LIN {X 0,Y 450.155,Z 511.876,A -85,B 0,C 180,E1 -8846.56,E2 -8846.56} C_VEL
LIN {X 0,Y 446.595,Z 503.795,A -85,B 0,C 180,E1 -8847.024,E2 -8847.024} C_VEL
LIN {X 0,Y 446.473,Z 503.185,A -85,B 0,C 180,E1 -8847.064,E2 -8847.064} C_VEL
LIN {X 0,Y 446.432,Z 503.191,A -85,B 0,C 180,E1 -8850.25,E2 -8850.25} C_VEL
LIN {X 0,Y 446.45,Z 503.188,A -85,B 0,C 180,E1 -8853.454,E2 -8853.454} C_VEL
LIN {X 0,Y 446.414,Z 503.19,A -85,B 0,C 180,E1 -8856.745,E2 -8856.745} C_VEL
LIN {X 0,Y 446.46,Z 503.185,A -85,B 0,C 180,E1 -8859.525,E2 -8859.525} C_VEL
LIN {X 0,Y 446.434,Z 503.188,A -85,B 0,C 180,E1 -8862.605,E2 -8862.605} C_VEL
LIN {X 0,Y 446.457,Z 503.185,A -85,B 0,C 180,E1 -8865.104,E2 -8865.104} C_VEL
LIN {X 0,Y 446.434,Z 503.189,A -85,B 0,C 180,E1 -8868.609,E2 -8868.609} C_VEL
LIN {X 0,Y 446.465,Z 503.184,A -85,B 0,C 180,E1 -8870.975,E2 -8870.975} C_VEL
LIN {X 0,Y 446.425,Z 503.194,A -85,B 0,C 180,E1 -8874.374,E2 -8874.374} C_VEL
LIN {X 0,Y 446.428,Z 503.194,A -85,B 0,C 180,E1 -8877.638,E2 -8877.638} C_VEL
LIN {X 0,Y 446.454,Z 503.189,A -85,B 0,C 180,E1 -8880.79,E2 -8880.79} C_VEL
LIN {X 0,Y 446.603,Z 503.368,A -85,B 0,C 180,E1 -8884.357,E2 -8884.357} C_VEL
LIN {X 0,Y 446.829,Z 506.002,A -85,B 0,C 180,E1 -8885.861,E2 -8885.861} C_VEL
LIN {X 0,Y 446.728,Z 511.144,A -85,B 0,C 180,E1 -8888.786,E2 -8888.786} C_VEL
LIN {X 0,Y 446.692,Z 516.086,A -85,B 0,C 180,E1 -8891.658,E2 -8891.658} C_VEL
LIN {X 0,Y 446.583,Z 520.857,A -85,B 0,C 180,E1 -8894.482,E2 -8894.482} C_VEL
LIN {X 0,Y 446.532,Z 523.772,A -85,B 0,C 180,E1 -8896.223,E2 -8896.223} C_VEL
LIN {X 0,Y 446.518,Z 525.315,A -85,B 0,C 180,E1 -8896.662,E2 -8896.662} C_VEL
LIN {X 0,Y 446.485,Z 527.885,A -85,B 0,C 180,E1 -8897.023,E2 -8897.023} C_VEL
LIN {X 0,Y 446.494,Z 532.862,A -85,B 0,C 180,E1 -8897.431,E2 -8897.431} C_VEL
LIN {X 0,Y 446.761,Z 538.729,A -85,B 0,C 180,E1 -8897.718,E2 -8897.718} C_VEL
LIN {X 0,Y 448.261,Z 548.9,A -85,B 0,C 180,E1 -8898.125,E2 -8898.125} C_VEL
LIN {X 0,Y 448.835,Z 550.834,A -85,B 0,C 180,E1 -8898.219,E2 -8898.219} C_VEL
LIN {X 0,Y 451.313,Z 559.337,A -85,B 0,C 180,E1 -8898.674,E2 -8898.674} C_VEL
LIN {X 0,Y 450.413,Z 575.184,A -85,B 0,C 180,E1 -8899.321,E2 -8899.321} C_VEL
LIN {X 0,Y 449.401,Z 589.936,A -85,B 0,C 180,E1 -8900.094,E2 -8900.094} C_VEL
LIN {X 0,Y 448.277,Z 603.783,A -85,B 0,C 180,E1 -8900.979,E2 -8900.979} C_VEL
LIN {X 0,Y 446.836,Z 619.369,A -85,B 0,C 180,E1 -8902.203,E2 -8902.203} C_VEL
LIN {X 0,Y 445.504,Z 632.325,A -85,B 0,C 180,E1 -8903.432,E2 -8903.432} C_VEL
LIN {X 0,Y 444.217,Z 644.41,A -85,B 0,C 180,E1 -8904.78,E2 -8904.78} C_VEL
LIN {X 0,Y 442.907,Z 656.466,A -85,B 0,C 180,E1 -8906.36,E2 -8906.36} C_VEL
LIN {X 0,Y 441.78,Z 666.782,A -85,B 0,C 180,E1 -8907.948,E2 -8907.948} C_VEL
LIN {X 0,Y 440.691,Z 676.755,A -85,B 0,C 180,E1 -8909.771,E2 -8909.771} C_VEL
LIN {X 0,Y 439.993,Z 684.187,A -85,B 0,C 180,E1 -8911.372,E2 -8911.372} C_VEL
LIN {X 0,Y 439.339,Z 691.448,A -85,B 0,C 180,E1 -8913.209,E2 -8913.209} C_VEL
LIN {X 0,Y 438.864,Z 698.729,A -85,B 0,C 180,E1 -8915.513,E2 -8915.513} C_VEL
LIN {X 0,Y 438.632,Z 703.269,A -85,B 0,C 180,E1 -8917.363,E2 -8917.363} C_VEL
LIN {X 0,Y 438.377,Z 706.848,A -85,B 0,C 180,E1 -8919.224,E2 -8919.224} C_VEL
LIN {X 0,Y 438.327,Z 709.385,A -85,B 0,C 180,E1 -8921.092,E2 -8921.092} C_VEL
LIN {X 0,Y 438.225,Z 710.957,A -85,B 0,C 180,E1 -8922.974,E2 -8922.974} C_VEL
LIN {X 0,Y 438.204,Z 711.571,A -85,B 0,C 180,E1 -8924.868,E2 -8924.868} C_VEL
LIN {X 0,Y 438.165,Z 711.15,A -85,B 0,C 180,E1 -8926.78,E2 -8926.78} C_VEL
LIN {X 0,Y 438.249,Z 709.566,A -85,B 0,C 180,E1 -8928.886,E2 -8928.886} C_VEL
LIN {X 0,Y 438.342,Z 707.239,A -85,B 0,C 180,E1 -8930.653,E2 -8930.653} C_VEL
LIN {X 0,Y 438.597,Z 703.612,A -85,B 0,C 180,E1 -8932.616,E2 -8932.616} C_VEL
LIN {X 0,Y 438.891,Z 698.778,A -85,B 0,C 180,E1 -8934.602,E2 -8934.602} C_VEL
LIN {X 0,Y 439.358,Z 692.513,A -85,B 0,C 180,E1 -8936.607,E2 -8936.607} C_VEL
LIN {X 0,Y 439.992,Z 684.737,A -85,B 0,C 180,E1 -8938.631,E2 -8938.631} C_VEL
LIN {X 0,Y 440.894,Z 675.565,A -85,B 0,C 180,E1 -8940.595,E2 -8940.595} C_VEL
LIN {X 0,Y 441.839,Z 666.752,A -85,B 0,C 180,E1 -8942.194,E2 -8942.194} C_VEL
LIN {X 0,Y 443.121,Z 655.256,A -85,B 0,C 180,E1 -8943.957,E2 -8943.957} C_VEL
LIN {X 0,Y 444.545,Z 642.016,A -85,B 0,C 180,E1 -8945.658,E2 -8945.658} C_VEL
LIN {X 0,Y 446.007,Z 628.866,A -85,B 0,C 180,E1 -8947.064,E2 -8947.064} C_VEL
LIN {X 0,Y 447.418,Z 614.816,A -85,B 0,C 180,E1 -8948.325,E2 -8948.325} C_VEL
LIN {X 0,Y 448.686,Z 600.827,A -85,B 0,C 180,E1 -8949.372,E2 -8949.372} C_VEL
LIN {X 0,Y 449.83,Z 586.318,A -85,B 0,C 180,E1 -8950.27,E2 -8950.27} C_VEL
LIN {X 0,Y 450.93,Z 570.329,A -85,B 0,C 180,E1 -8951.057,E2 -8951.057} C_VEL
LIN {X 0,Y 451.396,Z 558.681,A -85,B 0,C 180,E1 -8951.513,E2 -8951.513} C_VEL
LIN {X 0,Y 447.422,Z 546.372,A -85,B 0,C 180,E1 -8952.201,E2 -8952.201} C_VEL
LIN {X 0,Y 440.677,Z 529.846,A -85,B 0,C 180,E1 -8953.077,E2 -8953.077} C_VEL
LIN {X 0,Y 439.565,Z 526.832,A -85,B 0,C 180,E1 -8953.229,E2 -8953.229} C_VEL
LIN {X 0,Y 439.698,Z 521.329,A -85,B 0,C 180,E1 -8956.583,E2 -8956.583} C_VEL
LIN {X 0,Y 439.823,Z 517.224,A -85,B 0,C 180,E1 -8959.069,E2 -8959.069} C_VEL
LIN {X 0,Y 439.901,Z 513.154,A -85,B 0,C 180,E1 -8961.519,E2 -8961.519} C_VEL
LIN {X 0,Y 439.979,Z 509.374,A -85,B 0,C 180,E1 -8963.77,E2 -8963.77} C_VEL
LIN {X 0,Y 439.715,Z 505.572,A -85,B 0,C 180,E1 -8965.985,E2 -8965.985} C_VEL
LIN {X 0,Y 439.39,Z 504.071,A -85,B 0,C 180,E1 -8966.949,E2 -8966.949} C_VEL
LIN {X 0,Y 439.389,Z 504.069,A -85,B 0,C 180,E1 -8970.274,E2 -8970.274} C_VEL
LIN {X 0,Y 439.425,Z 504.062,A -85,B 0,C 180,E1 -8973.587,E2 -8973.587} C_VEL
LIN {X 0,Y 439.38,Z 504.067,A -85,B 0,C 180,E1 -8976.429,E2 -8976.429} C_VEL
LIN {X 0,Y 439.384,Z 504.068,A -85,B 0,C 180,E1 -8979.396,E2 -8979.396} C_VEL
LIN {X 0,Y 439.422,Z 504.063,A -85,B 0,C 180,E1 -8982.309,E2 -8982.309} C_VEL
LIN {X 0,Y 439.438,Z 504.06,A -85,B 0,C 180,E1 -8985.173,E2 -8985.173} C_VEL
LIN {X 0,Y 439.498,Z 504.053,A -85,B 0,C 180,E1 -8988.001,E2 -8988.001} C_VEL
LIN {X 0,Y 439.537,Z 504.043,A -85,B 0,C 180,E1 -8991.726,E2 -8991.726} C_VEL
LIN {X 0,Y 439.619,Z 504.035,A -85,B 0,C 180,E1 -8994.495,E2 -8994.495} C_VEL
LIN {X 0,Y 439.626,Z 504.031,A -85,B 0,C 180,E1 -8998.167,E2 -8998.167} C_VEL
LIN {X 0,Y 439.754,Z 504.021,A -85,B 0,C 180,E1 -9000,E2 -9000} C_VEL
LIN {X 0,Y 439.647,Z 504.031,A -85,B 0,C 180,E1 -9002.748,E2 -9002.748} C_VEL
LIN {X 0,Y 439.607,Z 504.038,A -85,B 0,C 180,E1 -9006.425,E2 -9006.425} C_VEL
LIN {X 0,Y 439.491,Z 504.047,A -85,B 0,C 180,E1 -9009.201,E2 -9009.201} C_VEL
LIN {X 0,Y 439.493,Z 504.046,A -85,B 0,C 180,E1 -9012.727,E2 -9012.727} C_VEL
LIN {X 0,Y 439.435,Z 504.045,A -85,B 0,C 180,E1 -9016.349,E2 -9016.349} C_VEL
LIN {X 0,Y 439.423,Z 504.053,A -85,B 0,C 180,E1 -9019.625,E2 -9019.625} C_VEL
LIN {X 0,Y 439.366,Z 504.062,A -85,B 0,C 180,E1 -9022.575,E2 -9022.575} C_VEL
LIN {X 0,Y 439.401,Z 504.046,A -85,B 0,C 180,E1 -9025.585,E2 -9025.585} C_VEL
LIN {X 0,Y 439.414,Z 504.063,A -85,B 0,C 180,E1 -9028.673,E2 -9028.673} C_VEL
LIN {X 0,Y 439.372,Z 504.069,A -85,B 0,C 180,E1 -9032.034,E2 -9032.034} C_VEL
LIN {X 0,Y 439.386,Z 504.064,A -85,B 0,C 180,E1 -9035.341,E2 -9035.341} C_VEL
LIN {X 0,Y 439.391,Z 504.064,A -85,B 0,C 180,E1 -9038.594,E2 -9038.594} C_VEL
LIN {X 0,Y 439.425,Z 504.199,A -85,B 0,C 180,E1 -9040.749,E2 -9040.749} C_VEL
LIN {X 0,Y 441.305,Z 512.586,A -85,B 0,C 180,E1 -9043.757,E2 -9043.757} C_VEL
LIN {X 0,Y 443.373,Z 522.19,A -85,B 0,C 180,E1 -9047.033,E2 -9047.033} C_VEL
LIN {X 0,Y 444.482,Z 528.015,A -85,B 0,C 180,E1 -9048.937,E2 -9048.937} C_VEL
LIN {X 0,Y 444.326,Z 534.065,A -85,B 0,C 180,E1 -9050.753,E2 -9050.753} C_VEL
LIN {X 0,Y 443.528,Z 545.656,A -85,B 0,C 180,E1 -9054.108,E2 -9054.108} C_VEL
LIN {X 0,Y 442.749,Z 557.216,A -85,B 0,C 180,E1 -9057.338,E2 -9057.338} C_VEL
LIN {X 0,Y 441.923,Z 570.71,A -85,B 0,C 180,E1 -9061.006,E2 -9061.006} C_VEL
LIN {X 0,Y 441.695,Z 574.164,A -85,B 0,C 180,E1 -9061.932,E2 -9061.932} C_VEL
LIN {X 0,Y 447.617,Z 596.261,A -85,B 0,C 180,E1 -9062.818,E2 -9062.818} C_VEL
LIN {X 0,Y 451.098,Z 610.608,A -85,B 0,C 180,E1 -9063.501,E2 -9063.501} C_VEL
LIN {X 0,Y 450.151,Z 626.715,A -85,B 0,C 180,E1 -9064.141,E2 -9064.141} C_VEL
LIN {X 0,Y 448.858,Z 643.305,A -85,B 0,C 180,E1 -9064.993,E2 -9064.993} C_VEL
LIN {X 0,Y 447.49,Z 659.254,A -85,B 0,C 180,E1 -9066.024,E2 -9066.024} C_VEL
LIN {X 0,Y 446.086,Z 673.924,A -85,B 0,C 180,E1 -9067.174,E2 -9067.174} C_VEL
LIN {X 0,Y 444.736,Z 687.558,A -85,B 0,C 180,E1 -9068.445,E2 -9068.445} C_VEL
LIN {X 0,Y 443.475,Z 700.18,A -85,B 0,C 180,E1 -9069.839,E2 -9069.839} C_VEL
LIN {X 0,Y 442.164,Z 712.75,A -85,B 0,C 180,E1 -9071.466,E2 -9071.466} C_VEL
LIN {X 0,Y 441.22,Z 722.902,A -85,B 0,C 180,E1 -9072.999,E2 -9072.999} C_VEL
LIN {X 0,Y 440.324,Z 732.743,A -85,B 0,C 180,E1 -9074.732,E2 -9074.732} C_VEL
LIN {X 0,Y 439.596,Z 741.658,A -85,B 0,C 180,E1 -9076.597,E2 -9076.597} C_VEL
LIN {X 0,Y 439.076,Z 749.128,A -85,B 0,C 180,E1 -9078.46,E2 -9078.46} C_VEL
LIN {X 0,Y 438.661,Z 755.325,A -85,B 0,C 180,E1 -9080.316,E2 -9080.316} C_VEL
LIN {X 0,Y 438.495,Z 760.18,A -85,B 0,C 180,E1 -9082.171,E2 -9082.171} C_VEL
LIN {X 0,Y 438.394,Z 763.307,A -85,B 0,C 180,E1 -9083.685,E2 -9083.685} C_VEL
LIN {X 0,Y 438.286,Z 765.978,A -85,B 0,C 180,E1 -9085.402,E2 -9085.402} C_VEL
LIN {X 0,Y 438.282,Z 767.896,A -85,B 0,C 180,E1 -9087.244,E2 -9087.244} C_VEL
LIN {X 0,Y 438.226,Z 768.847,A -85,B 0,C 180,E1 -9089.082,E2 -9089.082} C_VEL
LIN {X 0,Y 438.226,Z 768.847,A -85,B 0,C 180,E1 -9090.92,E2 -9090.92} C_VEL
LIN {X 0,Y 438.282,Z 767.893,A -85,B 0,C 180,E1 -9092.758,E2 -9092.758} C_VEL
LIN {X 0,Y 438.287,Z 765.974,A -85,B 0,C 180,E1 -9094.6,E2 -9094.6} C_VEL
LIN {X 0,Y 438.418,Z 763.059,A -85,B 0,C 180,E1 -9096.444,E2 -9096.444} C_VEL
LIN {X 0,Y 438.535,Z 759.098,A -85,B 0,C 180,E1 -9098.294,E2 -9098.294} C_VEL
LIN {X 0,Y 438.71,Z 753.832,A -85,B 0,C 180,E1 -9100.15,E2 -9100.15} C_VEL
LIN {X 0,Y 439.198,Z 747.328,A -85,B 0,C 180,E1 -9102.007,E2 -9102.007} C_VEL
LIN {X 0,Y 439.752,Z 739.357,A -85,B 0,C 180,E1 -9103.871,E2 -9103.871} C_VEL
LIN {X 0,Y 440.586,Z 729.818,A -85,B 0,C 180,E1 -9105.735,E2 -9105.735} C_VEL
LIN {X 0,Y 441.45,Z 719.525,A -85,B 0,C 180,E1 -9107.438,E2 -9107.438} C_VEL
LIN {X 0,Y 442.487,Z 708.476,A -85,B 0,C 180,E1 -9109.003,E2 -9109.003} C_VEL
LIN {X 0,Y 443.699,Z 695.677,A -85,B 0,C 180,E1 -9110.546,E2 -9110.546} C_VEL
LIN {X 0,Y 445.098,Z 681.138,A -85,B 0,C 180,E1 -9112.025,E2 -9112.025} C_VEL
LIN {X 0,Y 446.476,Z 666.202,A -85,B 0,C 180,E1 -9113.298,E2 -9113.298} C_VEL
LIN {X 0,Y 447.827,Z 650.15,A -85,B 0,C 180,E1 -9114.434,E2 -9114.434} C_VEL
LIN {X 0,Y 449.261,Z 632.83,A -85,B 0,C 180,E1 -9115.419,E2 -9115.419} C_VEL
LIN {X 0,Y 450.375,Z 616.592,A -85,B 0,C 180,E1 -9116.155,E2 -9116.155} C_VEL
LIN {X 0,Y 450.617,Z 609.71,A -85,B 0,C 180,E1 -9116.429,E2 -9116.429} C_VEL
LIN {X 0,Y 446.065,Z 591.603,A -85,B 0,C 180,E1 -9117.299,E2 -9117.299} C_VEL
LIN {X 0,Y 441.305,Z 569.539,A -85,B 0,C 180,E1 -9118.175,E2 -9118.175} C_VEL
LIN {X 0,Y 441.748,Z 557.378,A -85,B 0,C 180,E1 -9121.169,E2 -9121.169} C_VEL
LIN {X 0,Y 442.142,Z 544.142,A -85,B 0,C 180,E1 -9124.532,E2 -9124.532} C_VEL
LIN {X 0,Y 442.565,Z 534.404,A -85,B 0,C 180,E1 -9127.118,E2 -9127.118} C_VEL
LIN {X 0,Y 443.037,Z 524.605,A -85,B 0,C 180,E1 -9129.895,E2 -9129.895} C_VEL
LIN {X 0,Y 442.696,Z 520.674,A -85,B 0,C 180,E1 -9131.139,E2 -9131.139} C_VEL
LIN {X 0,Y 441.448,Z 513.639,A -85,B 0,C 180,E1 -9133.692,E2 -9133.692} C_VEL
LIN {X 0,Y 440.452,Z 508.687,A -85,B 0,C 180,E1 -9135.893,E2 -9135.893} C_VEL
LIN {X 0,Y 439.43,Z 504.239,A -85,B 0,C 180,E1 -9138.57,E2 -9138.57} C_VEL
LIN {X 0,Y 439.386,Z 504.068,A -85,B 0,C 180,E1 -9141.607,E2 -9141.607} C_VEL
LIN {X 0,Y 439.402,Z 504.065,A -85,B 0,C 180,E1 -9144.845,E2 -9144.845} C_VEL
LIN {X 0,Y 439.374,Z 504.069,A -85,B 0,C 180,E1 -9148.14,E2 -9148.14} C_VEL
LIN {X 0,Y 439.434,Z 504.061,A -85,B 0,C 180,E1 -9151.599,E2 -9151.599} C_VEL
LIN {X 0,Y 439.421,Z 504.063,A -85,B 0,C 180,E1 -9152.387,E2 -9152.387} C_VEL
LIN {X 0,Y 440.516,Z 507.043,A -85,B 0,C 180,E1 -9152.569,E2 -9152.569} C_VEL
LIN {X 0,Y 446.024,Z 518.302,A -85,B 0,C 180,E1 -9153.371,E2 -9153.371} C_VEL
LIN {X 0,Y 449.995,Z 528.652,A -85,B 0,C 180,E1 -9154.069,E2 -9154.069} C_VEL
LIN {X 0,Y 450.431,Z 530.462,A -85,B 0,C 180,E1 -9154.184,E2 -9154.184} C_VEL
LIN {X 0,Y 449.563,Z 546.73,A -85,B 0,C 180,E1 -9154.952,E2 -9154.952} C_VEL
LIN {X 0,Y 448.392,Z 562.457,A -85,B 0,C 180,E1 -9155.877,E2 -9155.877} C_VEL
LIN {X 0,Y 447.292,Z 576.15,A -85,B 0,C 180,E1 -9156.871,E2 -9156.871} C_VEL
LIN {X 0,Y 446.14,Z 589.85,A -85,B 0,C 180,E1 -9158.054,E2 -9158.054} C_VEL
LIN {X 0,Y 444.907,Z 602.248,A -85,B 0,C 180,E1 -9159.313,E2 -9159.313} C_VEL
LIN {X 0,Y 443.843,Z 612.936,A -85,B 0,C 180,E1 -9160.578,E2 -9160.578} C_VEL
LIN {X 0,Y 442.707,Z 624.177,A -85,B 0,C 180,E1 -9162.141,E2 -9162.141} C_VEL
LIN {X 0,Y 441.682,Z 634.47,A -85,B 0,C 180,E1 -9163.832,E2 -9163.832} C_VEL
LIN {X 0,Y 440.75,Z 643.955,A -85,B 0,C 180,E1 -9165.691,E2 -9165.691} C_VEL
LIN {X 0,Y 440.064,Z 651.852,A -85,B 0,C 180,E1 -9167.55,E2 -9167.55} C_VEL
LIN {X 0,Y 439.461,Z 658.362,A -85,B 0,C 180,E1 -9169.403,E2 -9169.403} C_VEL
LIN {X 0,Y 439.057,Z 664.718,A -85,B 0,C 180,E1 -9171.717,E2 -9171.717} C_VEL
LIN {X 0,Y 438.809,Z 668.498,A -85,B 0,C 180,E1 -9173.563,E2 -9173.563} C_VEL
LIN {X 0,Y 438.609,Z 671.321,A -85,B 0,C 180,E1 -9175.405,E2 -9175.405} C_VEL
LIN {X 0,Y 438.529,Z 673.1,A -85,B 0,C 180,E1 -9177.245,E2 -9177.245} C_VEL
LIN {X 0,Y 438.445,Z 673.979,A -85,B 0,C 180,E1 -9179.082,E2 -9179.082} C_VEL
LIN {X 0,Y 438.432,Z 673.872,A -85,B 0,C 180,E1 -9180.919,E2 -9180.919} C_VEL
LIN {X 0,Y 438.527,Z 672.857,A -85,B 0,C 180,E1 -9182.756,E2 -9182.756} C_VEL
LIN {X 0,Y 438.58,Z 670.871,A -85,B 0,C 180,E1 -9184.596,E2 -9184.596} C_VEL
LIN {X 0,Y 438.77,Z 667.318,A -85,B 0,C 180,E1 -9186.74,E2 -9186.74} C_VEL
LIN {X 0,Y 438.973,Z 662.731,A -85,B 0,C 180,E1 -9188.749,E2 -9188.749} C_VEL
LIN {X 0,Y 439.245,Z 657.369,A -85,B 0,C 180,E1 -9190.603,E2 -9190.603} C_VEL
LIN {X 0,Y 439.811,Z 650.68,A -85,B 0,C 180,E1 -9192.458,E2 -9192.458} C_VEL
LIN {X 0,Y 440.454,Z 642.654,A -85,B 0,C 180,E1 -9194.32,E2 -9194.32} C_VEL
LIN {X 0,Y 441.227,Z 634.366,A -85,B 0,C 180,E1 -9195.948,E2 -9195.948} C_VEL
LIN {X 0,Y 442.149,Z 624.564,A -85,B 0,C 180,E1 -9197.579,E2 -9197.579} C_VEL
LIN {X 0,Y 443.238,Z 613.092,A -85,B 0,C 180,E1 -9199.209,E2 -9199.209} C_VEL
LIN {X 0,Y 444.544,Z 600.249,A -85,B 0,C 180,E1 -9200.75,E2 -9200.75} C_VEL
LIN {X 0,Y 445.85,Z 586.862,A -85,B 0,C 180,E1 -9202.108,E2 -9202.108} C_VEL
LIN {X 0,Y 447.029,Z 573.338,A -85,B 0,C 180,E1 -9203.267,E2 -9203.267} C_VEL
LIN {X 0,Y 448.267,Z 558.807,A -85,B 0,C 180,E1 -9204.3,E2 -9204.3} C_VEL
LIN {X 0,Y 449.287,Z 544.247,A -85,B 0,C 180,E1 -9205.16,E2 -9205.16} C_VEL
LIN {X 0,Y 450.169,Z 530.335,A -85,B 0,C 180,E1 -9205.83,E2 -9205.83} C_VEL
LIN {X 0,Y 445.202,Z 517.627,A -85,B 0,C 180,E1 -9206.658,E2 -9206.658} C_VEL
LIN {X 0,Y 439.48,Z 504.426,A -85,B 0,C 180,E1 -9207.46,E2 -9207.46} C_VEL
LIN {X 0,Y 439.429,Z 504.06,A -85,B 0,C 180,E1 -9207.493,E2 -9207.493} C_VEL
LIN {X 0,Y 439.366,Z 504.07,A -85,B 0,C 180,E1 -9210.789,E2 -9210.789} C_VEL
LIN {X 0,Y 439.393,Z 504.065,A -85,B 0,C 180,E1 -9214.044,E2 -9214.044} C_VEL
LIN {X 0,Y 439.362,Z 504.069,A -85,B 0,C 180,E1 -9216.889,E2 -9216.889} C_VEL
LIN {X 0,Y 439.407,Z 504.064,A -85,B 0,C 180,E1 -9219.849,E2 -9219.849} C_VEL
LIN {X 0,Y 439.387,Z 504.066,A -85,B 0,C 180,E1 -9222.627,E2 -9222.627} C_VEL
LIN {X 0,Y 439.405,Z 504.063,A -85,B 0,C 180,E1 -9225.271,E2 -9225.271} C_VEL
LIN {X 0,Y 439.394,Z 504.067,A -85,B 0,C 180,E1 -9228.743,E2 -9228.743} C_VEL
LIN {X 0,Y 439.383,Z 504.069,A -85,B 0,C 180,E1 -9231.607,E2 -9231.607} C_VEL
LIN {X 0,Y 439.405,Z 504.066,A -85,B 0,C 180,E1 -9234.844,E2 -9234.844} C_VEL
LIN {X 0,Y 439.379,Z 504.072,A -85,B 0,C 180,E1 -9238.139,E2 -9238.139} C_VEL
LIN {X 0,Y 439.438,Z 504.063,A -85,B 0,C 180,E1 -9241.598,E2 -9241.598} C_VEL
LIN {X 0,Y 439.488,Z 504.068,A -85,B 0,C 180,E1 -9244.05,E2 -9244.05} C_VEL
LIN {X 0,Y 439.794,Z 508.249,A -85,B 0,C 180,E1 -9246.452,E2 -9246.452} C_VEL
LIN {X 0,Y 439.736,Z 513.41,A -85,B 0,C 180,E1 -9249.413,E2 -9249.413} C_VEL
LIN {X 0,Y 439.67,Z 518.364,A -85,B 0,C 180,E1 -9252.319,E2 -9252.319} C_VEL
LIN {X 0,Y 439.552,Z 523.155,A -85,B 0,C 180,E1 -9255.177,E2 -9255.177} C_VEL
LIN {X 0,Y 439.538,Z 526.233,A -85,B 0,C 180,E1 -9257.034,E2 -9257.034} C_VEL
LIN {X 0,Y 441.53,Z 531.586,A -85,B 0,C 180,E1 -9257.266,E2 -9257.266} C_VEL
LIN {X 0,Y 447.872,Z 548.086,A -85,B 0,C 180,E1 -9258.077,E2 -9258.077} C_VEL
LIN {X 0,Y 448.835,Z 550.834,A -85,B 0,C 180,E1 -9258.219,E2 -9258.219} C_VEL
LIN {X 0,Y 449.245,Z 553.899,A -85,B 0,C 180,E1 -9258.341,E2 -9258.341} C_VEL
LIN {X 0,Y 448.43,Z 558.379,A -85,B 0,C 180,E1 -9258.444,E2 -9258.444} C_VEL
LIN {X 0,Y 444.726,Z 568.644,A -85,B 0,C 180,E1 -9258.638,E2 -9258.638} C_VEL
LIN {X 0,Y 444.296,Z 571.249,A -85,B 0,C 180,E1 -9258.737,E2 -9258.737} C_VEL
LIN {X 0,Y 443.27,Z 586.441,A -85,B 0,C 180,E1 -9259.494,E2 -9259.494} C_VEL
LIN {X 0,Y 442.042,Z 600.861,A -85,B 0,C 180,E1 -9260.389,E2 -9260.389} C_VEL
LIN {X 0,Y 440.639,Z 615.729,A -85,B 0,C 180,E1 -9261.515,E2 -9261.515} C_VEL
LIN {X 0,Y 439.241,Z 629.393,A -85,B 0,C 180,E1 -9262.76,E2 -9262.76} C_VEL
LIN {X 0,Y 437.9,Z 641.066,A -85,B 0,C 180,E1 -9264.011,E2 -9264.011} C_VEL
LIN {X 0,Y 436.67,Z 651.988,A -85,B 0,C 180,E1 -9265.383,E2 -9265.383} C_VEL
LIN {X 0,Y 435.445,Z 663.002,A -85,B 0,C 180,E1 -9266.992,E2 -9266.992} C_VEL
LIN {X 0,Y 434.184,Z 673.693,A -85,B 0,C 180,E1 -9268.84,E2 -9268.84} C_VEL
LIN {X 0,Y 433.247,Z 682.67,A -85,B 0,C 180,E1 -9270.696,E2 -9270.696} C_VEL
LIN {X 0,Y 432.589,Z 689.313,A -85,B 0,C 180,E1 -9272.327,E2 -9272.327} C_VEL
LIN {X 0,Y 432.094,Z 695.775,A -85,B 0,C 180,E1 -9274.196,E2 -9274.196} C_VEL
LIN {X 0,Y 431.68,Z 702.18,A -85,B 0,C 180,E1 -9276.543,E2 -9276.543} C_VEL
LIN {X 0,Y 431.421,Z 706.076,A -85,B 0,C 180,E1 -9278.43,E2 -9278.43} C_VEL
LIN {X 0,Y 431.233,Z 709.019,A -85,B 0,C 180,E1 -9280.326,E2 -9280.326} C_VEL
LIN {X 0,Y 431.22,Z 710.935,A -85,B 0,C 180,E1 -9282.231,E2 -9282.231} C_VEL
LIN {X 0,Y 431.09,Z 711.9,A -85,B 0,C 180,E1 -9284.154,E2 -9284.154} C_VEL
LIN {X 0,Y 431.1,Z 711.888,A -85,B 0,C 180,E1 -9286.088,E2 -9286.088} C_VEL
LIN {X 0,Y 431.132,Z 710.828,A -85,B 0,C 180,E1 -9288.041,E2 -9288.041} C_VEL
LIN {X 0,Y 431.219,Z 708.784,A -85,B 0,C 180,E1 -9290.013,E2 -9290.013} C_VEL
LIN {X 0,Y 431.463,Z 705.545,A -85,B 0,C 180,E1 -9292.001,E2 -9292.001} C_VEL
LIN {X 0,Y 431.733,Z 701.145,A -85,B 0,C 180,E1 -9294.013,E2 -9294.013} C_VEL
LIN {X 0,Y 432.182,Z 695.469,A -85,B 0,C 180,E1 -9296.043,E2 -9296.043} C_VEL
LIN {X 0,Y 432.799,Z 688.302,A -85,B 0,C 180,E1 -9298.092,E2 -9298.092} C_VEL
LIN {X 0,Y 433.68,Z 679.444,A -85,B 0,C 180,E1 -9300.155,E2 -9300.155} C_VEL
LIN {X 0,Y 434.694,Z 670.095,A -85,B 0,C 180,E1 -9301.969,E2 -9301.969} C_VEL
LIN {X 0,Y 436.003,Z 658.98,A -85,B 0,C 180,E1 -9303.786,E2 -9303.786} C_VEL
LIN {X 0,Y 437.317,Z 647.707,A -85,B 0,C 180,E1 -9305.347,E2 -9305.347} C_VEL
LIN {X 0,Y 438.781,Z 635.463,A -85,B 0,C 180,E1 -9306.787,E2 -9306.787} C_VEL
LIN {X 0,Y 440.202,Z 622.509,A -85,B 0,C 180,E1 -9308.071,E2 -9308.071} C_VEL
LIN {X 0,Y 441.566,Z 608.746,A -85,B 0,C 180,E1 -9309.223,E2 -9309.223} C_VEL
LIN {X 0,Y 442.892,Z 594.051,A -85,B 0,C 180,E1 -9310.243,E2 -9310.243} C_VEL
LIN {X 0,Y 444.059,Z 579.672,A -85,B 0,C 180,E1 -9311.055,E2 -9311.055} C_VEL
LIN {X 0,Y 445.065,Z 563.239,A -85,B 0,C 180,E1 -9311.777,E2 -9311.777} C_VEL
LIN {X 0,Y 445.071,Z 560.384,A -85,B 0,C 180,E1 -9311.893,E2 -9311.893} C_VEL
LIN {X 0,Y 440.36,Z 546.175,A -85,B 0,C 180,E1 -9312.722,E2 -9312.722} C_VEL
LIN {X 0,Y 434.682,Z 532.439,A -85,B 0,C 180,E1 -9313.485,E2 -9313.485} C_VEL
LIN {X 0,Y 432.742,Z 528.017,A -85,B 0,C 180,E1 -9313.721,E2 -9313.721} C_VEL
LIN {X 0,Y 432.59,Z 527.264,A -85,B 0,C 180,E1 -9313.764,E2 -9313.764} C_VEL
LIN {X 0,Y 432.737,Z 521.997,A -85,B 0,C 180,E1 -9316.99,E2 -9316.99} C_VEL
LIN {X 0,Y 432.892,Z 517.519,A -85,B 0,C 180,E1 -9319.731,E2 -9319.731} C_VEL
LIN {X 0,Y 433.018,Z 511.947,A -85,B 0,C 180,E1 -9323.092,E2 -9323.092} C_VEL
LIN {X 0,Y 432.908,Z 508.112,A -85,B 0,C 180,E1 -9325.374,E2 -9325.374} C_VEL
LIN {X 0,Y 432.337,Z 504.949,A -85,B 0,C 180,E1 -9327.281,E2 -9327.281} C_VEL
LIN {X 0,Y 432.387,Z 504.943,A -85,B 0,C 180,E1 -9329.743,E2 -9329.743} C_VEL
LIN {X 0,Y 432.392,Z 504.938,A -85,B 0,C 180,E1 -9333.371,E2 -9333.371} C_VEL
LIN {X 0,Y 432.365,Z 504.944,A -85,B 0,C 180,E1 -9336.023,E2 -9336.023} C_VEL
LIN {X 0,Y 432.345,Z 504.943,A -85,B 0,C 180,E1 -9339.045,E2 -9339.045} C_VEL
LIN {X 0,Y 432.369,Z 504.943,A -85,B 0,C 180,E1 -9342.01,E2 -9342.01} C_VEL
LIN {X 0,Y 432.385,Z 504.939,A -85,B 0,C 180,E1 -9344.926,E2 -9344.926} C_VEL
LIN {X 0,Y 432.471,Z 504.928,A -85,B 0,C 180,E1 -9347.803,E2 -9347.803} C_VEL
LIN {X 0,Y 432.482,Z 504.922,A -85,B 0,C 180,E1 -9351.59,E2 -9351.59} C_VEL
LIN {X 0,Y 432.594,Z 504.91,A -85,B 0,C 180,E1 -9354.406,E2 -9354.406} C_VEL
LIN {X 0,Y 432.596,Z 504.907,A -85,B 0,C 180,E1 -9358.138,E2 -9358.138} C_VEL
LIN {X 0,Y 432.724,Z 504.896,A -85,B 0,C 180,E1 -9360,E2 -9360} C_VEL
LIN {X 0,Y 432.597,Z 504.909,A -85,B 0,C 180,E1 -9362.793,E2 -9362.793} C_VEL
LIN {X 0,Y 432.561,Z 504.915,A -85,B 0,C 180,E1 -9366.53,E2 -9366.53} C_VEL
LIN {X 0,Y 432.434,Z 504.927,A -85,B 0,C 180,E1 -9369.353,E2 -9369.353} C_VEL
LIN {X 0,Y 432.433,Z 504.925,A -85,B 0,C 180,E1 -9372.812,E2 -9372.812} C_VEL
LIN {X 0,Y 432.4,Z 504.917,A -85,B 0,C 180,E1 -9376.479,E2 -9376.479} C_VEL
LIN {X 0,Y 432.368,Z 504.936,A -85,B 0,C 180,E1 -9379.959,E2 -9379.959} C_VEL
LIN {X 0,Y 432.316,Z 504.938,A -85,B 0,C 180,E1 -9382.964,E2 -9382.964} C_VEL
LIN {X 0,Y 432.357,Z 504.931,A -85,B 0,C 180,E1 -9386.032,E2 -9386.032} C_VEL
LIN {X 0,Y 432.341,Z 504.946,A -85,B 0,C 180,E1 -9389.187,E2 -9389.187} C_VEL
LIN {X 0,Y 432.321,Z 504.947,A -85,B 0,C 180,E1 -9392.295,E2 -9392.295} C_VEL
LIN {X 0,Y 432.331,Z 504.945,A -85,B 0,C 180,E1 -9394.677,E2 -9394.677} C_VEL
LIN {X 0,Y 432.345,Z 504.942,A -85,B 0,C 180,E1 -9398.149,E2 -9398.149} C_VEL
LIN {X 0,Y 432.376,Z 505.044,A -85,B 0,C 180,E1 -9400.248,E2 -9400.248} C_VEL
LIN {X 0,Y 434.402,Z 514.157,A -85,B 0,C 180,E1 -9403.569,E2 -9403.569} C_VEL
LIN {X 0,Y 436.536,Z 524.022,A -85,B 0,C 180,E1 -9406.982,E2 -9406.982} C_VEL
LIN {X 0,Y 437.646,Z 530.162,A -85,B 0,C 180,E1 -9409.004,E2 -9409.004} C_VEL
LIN {X 0,Y 437.398,Z 536.16,A -85,B 0,C 180,E1 -9410.819,E2 -9410.819} C_VEL
LIN {X 0,Y 436.603,Z 547.258,A -85,B 0,C 180,E1 -9414.076,E2 -9414.076} C_VEL
LIN {X 0,Y 435.739,Z 559.013,A -85,B 0,C 180,E1 -9417.408,E2 -9417.408} C_VEL
LIN {X 0,Y 434.919,Z 572.014,A -85,B 0,C 180,E1 -9421.003,E2 -9421.003} C_VEL
LIN {X 0,Y 434.817,Z 573.58,A -85,B 0,C 180,E1 -9421.431,E2 -9421.431} C_VEL
LIN {X 0,Y 441.108,Z 597.306,A -85,B 0,C 180,E1 -9422.43,E2 -9422.43} C_VEL
LIN {X 0,Y 444.578,Z 611.784,A -85,B 0,C 180,E1 -9423.151,E2 -9423.151} C_VEL
LIN {X 0,Y 443.532,Z 628.476,A -85,B 0,C 180,E1 -9423.853,E2 -9423.853} C_VEL
LIN {X 0,Y 442.224,Z 644.05,A -85,B 0,C 180,E1 -9424.687,E2 -9424.687} C_VEL
LIN {X 0,Y 440.755,Z 660.103,A -85,B 0,C 180,E1 -9425.759,E2 -9425.759} C_VEL
LIN {X 0,Y 439.292,Z 674.487,A -85,B 0,C 180,E1 -9426.925,E2 -9426.925} C_VEL
LIN {X 0,Y 437.79,Z 689.017,A -85,B 0,C 180,E1 -9428.333,E2 -9428.333} C_VEL
LIN {X 0,Y 436.474,Z 701.391,A -85,B 0,C 180,E1 -9429.747,E2 -9429.747} C_VEL
LIN {X 0,Y 435.129,Z 713.666,A -85,B 0,C 180,E1 -9431.399,E2 -9431.399} C_VEL
LIN {X 0,Y 434.116,Z 724.16,A -85,B 0,C 180,E1 -9433.059,E2 -9433.059} C_VEL
LIN {X 0,Y 433.233,Z 733.216,A -85,B 0,C 180,E1 -9434.717,E2 -9434.717} C_VEL
LIN {X 0,Y 432.51,Z 741.976,A -85,B 0,C 180,E1 -9436.613,E2 -9436.613} C_VEL
LIN {X 0,Y 432.037,Z 748.418,A -85,B 0,C 180,E1 -9438.269,E2 -9438.269} C_VEL
LIN {X 0,Y 431.578,Z 754.613,A -85,B 0,C 180,E1 -9440.156,E2 -9440.156} C_VEL
LIN {X 0,Y 431.394,Z 760.648,A -85,B 0,C 180,E1 -9442.512,E2 -9442.512} C_VEL
LIN {X 0,Y 431.237,Z 764.178,A -85,B 0,C 180,E1 -9444.389,E2 -9444.389} C_VEL
LIN {X 0,Y 431.141,Z 766.738,A -85,B 0,C 180,E1 -9446.262,E2 -9446.262} C_VEL
LIN {X 0,Y 431.191,Z 768.197,A -85,B 0,C 180,E1 -9448.133,E2 -9448.133} C_VEL
LIN {X 0,Y 431.117,Z 768.732,A -85,B 0,C 180,E1 -9450.001,E2 -9450.001} C_VEL
LIN {X 0,Y 431.191,Z 768.189,A -85,B 0,C 180,E1 -9451.869,E2 -9451.869} C_VEL
LIN {X 0,Y 431.141,Z 766.714,A -85,B 0,C 180,E1 -9453.739,E2 -9453.739} C_VEL
LIN {X 0,Y 431.257,Z 764.133,A -85,B 0,C 180,E1 -9455.612,E2 -9455.612} C_VEL
LIN {X 0,Y 431.414,Z 760.561,A -85,B 0,C 180,E1 -9457.489,E2 -9457.489} C_VEL
LIN {X 0,Y 431.553,Z 755.771,A -85,B 0,C 180,E1 -9459.373,E2 -9459.373} C_VEL
LIN {X 0,Y 431.906,Z 749.813,A -85,B 0,C 180,E1 -9461.261,E2 -9461.261} C_VEL
LIN {X 0,Y 432.444,Z 742.549,A -85,B 0,C 180,E1 -9463.152,E2 -9463.152} C_VEL
LIN {X 0,Y 433.094,Z 733.749,A -85,B 0,C 180,E1 -9465.049,E2 -9465.049} C_VEL
LIN {X 0,Y 433.951,Z 724.684,A -85,B 0,C 180,E1 -9466.707,E2 -9466.707} C_VEL
LIN {X 0,Y 434.904,Z 714.084,A -85,B 0,C 180,E1 -9468.369,E2 -9468.369} C_VEL
LIN {X 0,Y 436.158,Z 701.686,A -85,B 0,C 180,E1 -9470.025,E2 -9470.025} C_VEL
LIN {X 0,Y 437.485,Z 688.617,A -85,B 0,C 180,E1 -9471.502,E2 -9471.502} C_VEL
LIN {X 0,Y 438.874,Z 674.607,A -85,B 0,C 180,E1 -9472.852,E2 -9472.852} C_VEL
LIN {X 0,Y 440.255,Z 660.216,A -85,B 0,C 180,E1 -9474.022,E2 -9474.022} C_VEL
LIN {X 0,Y 441.681,Z 644.106,A -85,B 0,C 180,E1 -9475.11,E2 -9475.11} C_VEL
LIN {X 0,Y 443.048,Z 627.986,A -85,B 0,C 180,E1 -9475.99,E2 -9475.99} C_VEL
LIN {X 0,Y 444.086,Z 611.413,A -85,B 0,C 180,E1 -9476.716,E2 -9476.716} C_VEL
LIN {X 0,Y 439.132,Z 590.647,A -85,B 0,C 180,E1 -9477.775,E2 -9477.775} C_VEL
LIN {X 0,Y 434.852,Z 571.012,A -85,B 0,C 180,E1 -9478.607,E2 -9478.607} C_VEL
LIN {X 0,Y 434.317,Z 567.994,A -85,B 0,C 180,E1 -9478.752,E2 -9478.752} C_VEL
LIN {X 0,Y 434.786,Z 555.299,A -85,B 0,C 180,E1 -9481.964,E2 -9481.964} C_VEL
LIN {X 0,Y 435.357,Z 541.712,A -85,B 0,C 180,E1 -9485.532,E2 -9485.532} C_VEL
LIN {X 0,Y 435.775,Z 531.517,A -85,B 0,C 180,E1 -9488.383,E2 -9488.383} C_VEL
LIN {X 0,Y 436.131,Z 525.633,A -85,B 0,C 180,E1 -9490.135,E2 -9490.135} C_VEL
LIN {X 0,Y 435.727,Z 521.829,A -85,B 0,C 180,E1 -9491.4,E2 -9491.4} C_VEL
LIN {X 0,Y 434.826,Z 516.613,A -85,B 0,C 180,E1 -9493.338,E2 -9493.338} C_VEL
LIN {X 0,Y 433.753,Z 511.023,A -85,B 0,C 180,E1 -9495.836,E2 -9495.836} C_VEL
LIN {X 0,Y 432.779,Z 506.867,A -85,B 0,C 180,E1 -9498.332,E2 -9498.332} C_VEL
LIN {X 0,Y 432.373,Z 504.941,A -85,B 0,C 180,E1 -9500.029,E2 -9500.029} C_VEL
LIN {X 0,Y 432.317,Z 504.948,A -85,B 0,C 180,E1 -9503.023,E2 -9503.023} C_VEL
LIN {X 0,Y 432.361,Z 504.942,A -85,B 0,C 180,E1 -9505.997,E2 -9505.997} C_VEL
LIN {X 0,Y 432.349,Z 504.944,A -85,B 0,C 180,E1 -9509.49,E2 -9509.49} C_VEL
LIN {X 0,Y 432.407,Z 504.937,A -85,B 0,C 180,E1 -9511.792,E2 -9511.792} C_VEL
LIN {X 0,Y 433.481,Z 507.906,A -85,B 0,C 180,E1 -9512,E2 -9512} C_VEL
LIN {X 0,Y 438.475,Z 517.712,A -85,B 0,C 180,E1 -9512.762,E2 -9512.762} C_VEL
LIN {X 0,Y 442.941,Z 528.615,A -85,B 0,C 180,E1 -9513.557,E2 -9513.557} C_VEL
LIN {X 0,Y 444.058,Z 531.924,A -85,B 0,C 180,E1 -9513.79,E2 -9513.79} C_VEL
LIN {X 0,Y 443.23,Z 547.896,A -85,B 0,C 180,E1 -9514.571,E2 -9514.571} C_VEL
LIN {X 0,Y 441.978,Z 563.437,A -85,B 0,C 180,E1 -9515.506,E2 -9515.506} C_VEL
LIN {X 0,Y 440.718,Z 578.581,A -85,B 0,C 180,E1 -9516.63,E2 -9516.63} C_VEL
LIN {X 0,Y 439.475,Z 592.085,A -85,B 0,C 180,E1 -9517.84,E2 -9517.84} C_VEL
LIN {X 0,Y 438.19,Z 604.143,A -85,B 0,C 180,E1 -9519.106,E2 -9519.106} C_VEL
LIN {X 0,Y 437.011,Z 615.574,A -85,B 0,C 180,E1 -9520.507,E2 -9520.507} C_VEL
LIN {X 0,Y 435.793,Z 626.994,A -85,B 0,C 180,E1 -9522.157,E2 -9522.157} C_VEL
LIN {X 0,Y 434.628,Z 637.905,A -85,B 0,C 180,E1 -9524.045,E2 -9524.045} C_VEL
LIN {X 0,Y 433.69,Z 646.962,A -85,B 0,C 180,E1 -9525.932,E2 -9525.932} C_VEL
LIN {X 0,Y 432.935,Z 654.441,A -85,B 0,C 180,E1 -9527.817,E2 -9527.817} C_VEL
LIN {X 0,Y 432.413,Z 660.585,A -85,B 0,C 180,E1 -9529.702,E2 -9529.702} C_VEL
LIN {X 0,Y 432.073,Z 665.563,A -85,B 0,C 180,E1 -9531.583,E2 -9531.583} C_VEL
LIN {X 0,Y 431.807,Z 669.348,A -85,B 0,C 180,E1 -9533.458,E2 -9533.458} C_VEL
LIN {X 0,Y 431.583,Z 672.168,A -85,B 0,C 180,E1 -9535.33,E2 -9535.33} C_VEL
LIN {X 0,Y 431.489,Z 673.937,A -85,B 0,C 180,E1 -9537.2,E2 -9537.2} C_VEL
LIN {X 0,Y 431.394,Z 674.795,A -85,B 0,C 180,E1 -9539.067,E2 -9539.067} C_VEL
LIN {X 0,Y 431.38,Z 674.68,A -85,B 0,C 180,E1 -9540.934,E2 -9540.934} C_VEL
LIN {X 0,Y 431.487,Z 673.628,A -85,B 0,C 180,E1 -9542.801,E2 -9542.801} C_VEL
LIN {X 0,Y 431.604,Z 672.769,A -85,B 0,C 180,E1 -9543.735,E2 -9543.735} C_VEL
LIN {X 0,Y 431.577,Z 670.243,A -85,B 0,C 180,E1 -9545.608,E2 -9545.608} C_VEL
LIN {X 0,Y 431.823,Z 666.758,A -85,B 0,C 180,E1 -9547.482,E2 -9547.482} C_VEL
LIN {X 0,Y 432.035,Z 662.159,A -85,B 0,C 180,E1 -9549.362,E2 -9549.362} C_VEL
LIN {X 0,Y 432.364,Z 656.416,A -85,B 0,C 180,E1 -9551.249,E2 -9551.249} C_VEL
LIN {X 0,Y 433.05,Z 649.322,A -85,B 0,C 180,E1 -9553.157,E2 -9553.157} C_VEL
LIN {X 0,Y 433.758,Z 640.938,A -85,B 0,C 180,E1 -9555.026,E2 -9555.026} C_VEL
LIN {X 0,Y 434.648,Z 632.132,A -85,B 0,C 180,E1 -9556.679,E2 -9556.679} C_VEL
LIN {X 0,Y 435.641,Z 621.881,A -85,B 0,C 180,E1 -9558.336,E2 -9558.336} C_VEL
LIN {X 0,Y 436.912,Z 609.812,A -85,B 0,C 180,E1 -9559.988,E2 -9559.988} C_VEL
LIN {X 0,Y 438.361,Z 595.912,A -85,B 0,C 180,E1 -9561.583,E2 -9561.583} C_VEL
LIN {X 0,Y 439.738,Z 581.875,A -85,B 0,C 180,E1 -9562.928,E2 -9562.928} C_VEL
LIN {X 0,Y 440.933,Z 568.795,A -85,B 0,C 180,E1 -9563.982,E2 -9563.982} C_VEL
LIN {X 0,Y 442.091,Z 553.485,A -85,B 0,C 180,E1 -9565.022,E2 -9565.022} C_VEL
LIN {X 0,Y 443.3,Z 537.381,A -85,B 0,C 180,E1 -9565.896,E2 -9565.896} C_VEL
LIN {X 0,Y 443.468,Z 531.483,A -85,B 0,C 180,E1 -9566.182,E2 -9566.182} C_VEL
LIN {X 0,Y 437.221,Z 516.147,A -85,B 0,C 180,E1 -9567.22,E2 -9567.22} C_VEL
LIN {X 0,Y 432.548,Z 505.754,A -85,B 0,C 180,E1 -9567.864,E2 -9567.864} C_VEL
LIN {X 0,Y 432.413,Z 504.932,A -85,B 0,C 180,E1 -9567.928,E2 -9567.928} C_VEL
LIN {X 0,Y 432.326,Z 504.947,A -85,B 0,C 180,E1 -9571.346,E2 -9571.346} C_VEL
LIN {X 0,Y 432.346,Z 504.946,A -85,B 0,C 180,E1 -9574.677,E2 -9574.677} C_VEL
LIN {X 0,Y 432.35,Z 504.942,A -85,B 0,C 180,E1 -9578.149,E2 -9578.149} C_VEL
LIN {X 0,Y 432.338,Z 504.946,A -85,B 0,C 180,E1 -9581.602,E2 -9581.602} C_VEL
LIN {X 0,Y 432.339,Z 504.945,A -85,B 0,C 180,E1 -9584.347,E2 -9584.347} C_VEL
LIN {X 0,Y 432.325,Z 504.945,A -85,B 0,C 180,E1 -9587.016,E2 -9587.016} C_VEL
LIN {X 0,Y 432.347,Z 504.943,A -85,B 0,C 180,E1 -9589.819,E2 -9589.819} C_VEL
LIN {X 0,Y 432.312,Z 504.948,A -85,B 0,C 180,E1 -9593.022,E2 -9593.022} C_VEL
LIN {X 0,Y 432.365,Z 504.945,A -85,B 0,C 180,E1 -9595.996,E2 -9595.996} C_VEL
LIN {X 0,Y 432.353,Z 504.947,A -85,B 0,C 180,E1 -9599.489,E2 -9599.489} C_VEL
LIN {X 0,Y 432.405,Z 504.937,A -85,B 0,C 180,E1 -9602.928,E2 -9602.928} C_VEL
LIN {X 0,Y 432.463,Z 505.014,A -85,B 0,C 180,E1 -9603.879,E2 -9603.879} C_VEL
LIN {X 0,Y 432.792,Z 508.795,A -85,B 0,C 180,E1 -9606.047,E2 -9606.047} C_VEL
LIN {X 0,Y 432.738,Z 514.003,A -85,B 0,C 180,E1 -9609.065,E2 -9609.065} C_VEL
LIN {X 0,Y 432.673,Z 519.036,A -85,B 0,C 180,E1 -9612.023,E2 -9612.023} C_VEL
LIN {X 0,Y 432.566,Z 523.923,A -85,B 0,C 180,E1 -9614.932,E2 -9614.932} C_VEL
LIN {X 0,Y 432.518,Z 526.626,A -85,B 0,C 180,E1 -9616.562,E2 -9616.562} C_VEL
LIN {X 0,Y 434.851,Z 532.693,A -85,B 0,C 180,E1 -9616.842,E2 -9616.842} C_VEL
LIN {X 0,Y 441.14,Z 549.032,A -85,B 0,C 180,E1 -9617.671,E2 -9617.671} C_VEL
LIN {X 0,Y 444.809,Z 560.472,A -85,B 0,C 180,E1 -9618.302,E2 -9618.302} C_VEL
LIN {X 0,Y 444.296,Z 571.249,A -85,B 0,C 180,E1 -9618.737,E2 -9618.737} C_VEL
LIN {X 0,Y 443.325,Z 577.004,A -85,B 0,C 180,E1 -9618.963,E2 -9618.963} C_VEL
LIN {X 0,Y 437.354,Z 593.09,A -85,B 0,C 180,E1 -9619.547,E2 -9619.547} C_VEL
LIN {X 0,Y 435.923,Z 598.391,A -85,B 0,C 180,E1 -9619.825,E2 -9619.825} C_VEL
LIN {X 0,Y 435.669,Z 600.092,A -85,B 0,C 180,E1 -9619.937,E2 -9619.937} C_VEL
LIN {X 0,Y 434.24,Z 614.741,A -85,B 0,C 180,E1 -9621.037,E2 -9621.037} C_VEL
LIN {X 0,Y 432.757,Z 628.682,A -85,B 0,C 180,E1 -9622.299,E2 -9622.299} C_VEL
LIN {X 0,Y 431.244,Z 641.467,A -85,B 0,C 180,E1 -9623.683,E2 -9623.683} C_VEL
LIN {X 0,Y 429.939,Z 652.402,A -85,B 0,C 180,E1 -9625.076,E2 -9625.076} C_VEL
LIN {X 0,Y 428.656,Z 663.42,A -85,B 0,C 180,E1 -9626.709,E2 -9626.709} C_VEL
LIN {X 0,Y 427.338,Z 674.129,A -85,B 0,C 180,E1 -9628.585,E2 -9628.585} C_VEL
LIN {X 0,Y 426.318,Z 683.128,A -85,B 0,C 180,E1 -9630.471,E2 -9630.471} C_VEL
LIN {X 0,Y 425.534,Z 690.648,A -85,B 0,C 180,E1 -9632.365,E2 -9632.365} C_VEL
LIN {X 0,Y 425.027,Z 696.924,A -85,B 0,C 180,E1 -9634.266,E2 -9634.266} C_VEL
LIN {X 0,Y 424.651,Z 702.06,A -85,B 0,C 180,E1 -9636.174,E2 -9636.174} C_VEL
LIN {X 0,Y 424.471,Z 705.217,A -85,B 0,C 180,E1 -9637.61,E2 -9637.61} C_VEL
LIN {X 0,Y 424.224,Z 708.475,A -85,B 0,C 180,E1 -9639.535,E2 -9639.535} C_VEL
LIN {X 0,Y 424.158,Z 710.793,A -85,B 0,C 180,E1 -9641.467,E2 -9641.467} C_VEL
LIN {X 0,Y 424.053,Z 712.103,A -85,B 0,C 180,E1 -9643.415,E2 -9643.415} C_VEL
LIN {X 0,Y 424.027,Z 712.451,A -85,B 0,C 180,E1 -9645.377,E2 -9645.377} C_VEL
LIN {X 0,Y 424.012,Z 711.809,A -85,B 0,C 180,E1 -9647.357,E2 -9647.357} C_VEL
LIN {X 0,Y 424.11,Z 710.095,A -85,B 0,C 180,E1 -9649.354,E2 -9649.354} C_VEL
LIN {X 0,Y 424.308,Z 707.359,A -85,B 0,C 180,E1 -9651.369,E2 -9651.369} C_VEL
LIN {X 0,Y 424.541,Z 703.385,A -85,B 0,C 180,E1 -9653.408,E2 -9653.408} C_VEL
LIN {X 0,Y 424.976,Z 698.168,A -85,B 0,C 180,E1 -9655.464,E2 -9655.464} C_VEL
LIN {X 0,Y 425.583,Z 691.589,A -85,B 0,C 180,E1 -9657.54,E2 -9657.54} C_VEL
LIN {X 0,Y 426.393,Z 683.433,A -85,B 0,C 180,E1 -9659.633,E2 -9659.633} C_VEL
LIN {X 0,Y 427.341,Z 675.1,A -85,B 0,C 180,E1 -9661.405,E2 -9661.405} C_VEL
LIN {X 0,Y 428.603,Z 664.825,A -85,B 0,C 180,E1 -9663.251,E2 -9663.251} C_VEL
LIN {X 0,Y 430.001,Z 654.045,A -85,B 0,C 180,E1 -9664.891,E2 -9664.891} C_VEL
LIN {X 0,Y 431.423,Z 641.816,A -85,B 0,C 180,E1 -9666.482,E2 -9666.482} C_VEL
LIN {X 0,Y 433.087,Z 628.521,A -85,B 0,C 180,E1 -9667.929,E2 -9667.929} C_VEL
LIN {X 0,Y 434.679,Z 614.059,A -85,B 0,C 180,E1 -9669.239,E2 -9669.239} C_VEL
LIN {X 0,Y 436.145,Z 599.127,A -85,B 0,C 180,E1 -9670.353,E2 -9670.353} C_VEL
LIN {X 0,Y 437.373,Z 585.125,A -85,B 0,C 180,E1 -9671.208,E2 -9671.208} C_VEL
LIN {X 0,Y 438.479,Z 569.364,A -85,B 0,C 180,E1 -9671.982,E2 -9671.982} C_VEL
LIN {X 0,Y 438.777,Z 562.116,A -85,B 0,C 180,E1 -9672.285,E2 -9672.285} C_VEL
LIN {X 0,Y 433.683,Z 546.926,A -85,B 0,C 180,E1 -9673.208,E2 -9673.208} C_VEL
LIN {X 0,Y 427.167,Z 531.428,A -85,B 0,C 180,E1 -9674.106,E2 -9674.106} C_VEL
LIN {X 0,Y 425.841,Z 528.548,A -85,B 0,C 180,E1 -9674.271,E2 -9674.271} C_VEL
LIN {X 0,Y 425.648,Z 527.686,A -85,B 0,C 180,E1 -9674.34,E2 -9674.34} C_VEL
LIN {X 0,Y 425.874,Z 521.809,A -85,B 0,C 180,E1 -9677.952,E2 -9677.952} C_VEL
LIN {X 0,Y 425.985,Z 516.591,A -85,B 0,C 180,E1 -9681.175,E2 -9681.175} C_VEL
LIN {X 0,Y 426.088,Z 512.112,A -85,B 0,C 180,E1 -9683.919,E2 -9683.919} C_VEL
LIN {X 0,Y 425.88,Z 508.735,A -85,B 0,C 180,E1 -9685.869,E2 -9685.869} C_VEL
LIN {X 0,Y 425.283,Z 505.83,A -85,B 0,C 180,E1 -9687.742,E2 -9687.742} C_VEL
LIN {X 0,Y 425.33,Z 505.819,A -85,B 0,C 180,E1 -9691.367,E2 -9691.367} C_VEL
LIN {X 0,Y 425.292,Z 505.823,A -85,B 0,C 180,E1 -9694.554,E2 -9694.554} C_VEL
LIN {X 0,Y 425.279,Z 505.827,A -85,B 0,C 180,E1 -9697.66,E2 -9697.66} C_VEL
LIN {X 0,Y 425.355,Z 505.813,A -85,B 0,C 180,E1 -9700.703,E2 -9700.703} C_VEL
LIN {X 0,Y 425.378,Z 505.807,A -85,B 0,C 180,E1 -9703.687,E2 -9703.687} C_VEL
LIN {X 0,Y 425.42,Z 505.807,A -85,B 0,C 180,E1 -9707.598,E2 -9707.598} C_VEL
LIN {X 0,Y 425.432,Z 505.801,A -85,B 0,C 180,E1 -9711.449,E2 -9711.449} C_VEL
LIN {X 0,Y 425.569,Z 505.785,A -85,B 0,C 180,E1 -9714.313,E2 -9714.313} C_VEL
LIN {X 0,Y 425.566,Z 505.783,A -85,B 0,C 180,E1 -9718.107,E2 -9718.107} C_VEL
LIN {X 0,Y 425.694,Z 505.772,A -85,B 0,C 180,E1 -9720,E2 -9720} C_VEL
LIN {X 0,Y 425.548,Z 505.787,A -85,B 0,C 180,E1 -9722.839,E2 -9722.839} C_VEL
LIN {X 0,Y 425.52,Z 505.792,A -85,B 0,C 180,E1 -9726.639,E2 -9726.639} C_VEL
LIN {X 0,Y 425.393,Z 505.804,A -85,B 0,C 180,E1 -9729.509,E2 -9729.509} C_VEL
LIN {X 0,Y 425.393,Z 505.803,A -85,B 0,C 180,E1 -9732.91,E2 -9732.91} C_VEL
LIN {X 0,Y 425.349,Z 505.792,A -85,B 0,C 180,E1 -9736.605,E2 -9736.605} C_VEL
LIN {X 0,Y 425.35,Z 505.805,A -85,B 0,C 180,E1 -9739.649,E2 -9739.649} C_VEL
LIN {X 0,Y 425.323,Z 505.813,A -85,B 0,C 180,E1 -9742.336,E2 -9742.336} C_VEL
LIN {X 0,Y 425.288,Z 505.799,A -85,B 0,C 180,E1 -9745.445,E2 -9745.445} C_VEL
LIN {X 0,Y 425.327,Z 505.817,A -85,B 0,C 180,E1 -9748.632,E2 -9748.632} C_VEL
LIN {X 0,Y 425.262,Z 505.826,A -85,B 0,C 180,E1 -9751.927,E2 -9751.927} C_VEL
LIN {X 0,Y 425.29,Z 505.82,A -85,B 0,C 180,E1 -9755.336,E2 -9755.336} C_VEL
LIN {X 0,Y 425.306,Z 505.819,A -85,B 0,C 180,E1 -9759.047,E2 -9759.047} C_VEL
LIN {X 0,Y 425.347,Z 505.954,A -85,B 0,C 180,E1 -9759.757,E2 -9759.757} C_VEL
LIN {X 0,Y 427.304,Z 514.797,A -85,B 0,C 180,E1 -9763.044,E2 -9763.044} C_VEL
LIN {X 0,Y 429.164,Z 523.442,A -85,B 0,C 180,E1 -9766.099,E2 -9766.099} C_VEL
LIN {X 0,Y 430.663,Z 530.979,A -85,B 0,C 180,E1 -9768.648,E2 -9768.648} C_VEL
LIN {X 0,Y 430.679,Z 535.564,A -85,B 0,C 180,E1 -9770.082,E2 -9770.082} C_VEL
LIN {X 0,Y 429.874,Z 546.111,A -85,B 0,C 180,E1 -9773.235,E2 -9773.235} C_VEL
LIN {X 0,Y 428.881,Z 558.974,A -85,B 0,C 180,E1 -9776.966,E2 -9776.966} C_VEL
LIN {X 0,Y 428.009,Z 571.485,A -85,B 0,C 180,E1 -9780.49,E2 -9780.49} C_VEL
LIN {X 0,Y 427.932,Z 573.059,A -85,B 0,C 180,E1 -9780.929,E2 -9780.929} C_VEL
LIN {X 0,Y 433.961,Z 595.903,A -85,B 0,C 180,E1 -9781.913,E2 -9781.913} C_VEL
LIN {X 0,Y 438.101,Z 613.116,A -85,B 0,C 180,E1 -9782.805,E2 -9782.805} C_VEL
LIN {X 0,Y 436.921,Z 630.132,A -85,B 0,C 180,E1 -9783.555,E2 -9783.555} C_VEL
LIN {X 0,Y 435.402,Z 646.765,A -85,B 0,C 180,E1 -9784.494,E2 -9784.494} C_VEL
LIN {X 0,Y 433.878,Z 662.463,A -85,B 0,C 180,E1 -9785.605,E2 -9785.605} C_VEL
LIN {X 0,Y 432.395,Z 676.334,A -85,B 0,C 180,E1 -9786.788,E2 -9786.788} C_VEL
LIN {X 0,Y 430.857,Z 690.092,A -85,B 0,C 180,E1 -9788.177,E2 -9788.177} C_VEL
LIN {X 0,Y 429.462,Z 702.497,A -85,B 0,C 180,E1 -9789.652,E2 -9789.652} C_VEL
LIN {X 0,Y 428.088,Z 714.557,A -85,B 0,C 180,E1 -9791.33,E2 -9791.33} C_VEL
LIN {X 0,Y 426.902,Z 726.19,A -85,B 0,C 180,E1 -9793.257,E2 -9793.257} C_VEL
LIN {X 0,Y 425.918,Z 735.94,A -85,B 0,C 180,E1 -9795.182,E2 -9795.182} C_VEL
LIN {X 0,Y 425.267,Z 744.364,A -85,B 0,C 180,E1 -9797.17,E2 -9797.17} C_VEL
LIN {X 0,Y 424.75,Z 750.965,A -85,B 0,C 180,E1 -9799.032,E2 -9799.032} C_VEL
LIN {X 0,Y 424.423,Z 756.511,A -85,B 0,C 180,E1 -9800.95,E2 -9800.95} C_VEL
LIN {X 0,Y 424.318,Z 759.941,A -85,B 0,C 180,E1 -9802.387,E2 -9802.387} C_VEL
LIN {X 0,Y 424.174,Z 763.477,A -85,B 0,C 180,E1 -9804.296,E2 -9804.296} C_VEL
LIN {X 0,Y 424.086,Z 766.031,A -85,B 0,C 180,E1 -9806.2,E2 -9806.2} C_VEL
LIN {X 0,Y 424.148,Z 767.487,A -85,B 0,C 180,E1 -9808.102,E2 -9808.102} C_VEL
LIN {X 0,Y 424.068,Z 768.003,A -85,B 0,C 180,E1 -9810.001,E2 -9810.001} C_VEL
LIN {X 0,Y 424.149,Z 767.45,A -85,B 0,C 180,E1 -9811.9,E2 -9811.9} C_VEL
LIN {X 0,Y 424.086,Z 765.941,A -85,B 0,C 180,E1 -9813.802,E2 -9813.802} C_VEL
LIN {X 0,Y 424.215,Z 763.341,A -85,B 0,C 180,E1 -9815.706,E2 -9815.706} C_VEL
LIN {X 0,Y 424.337,Z 759.718,A -85,B 0,C 180,E1 -9817.615,E2 -9817.615} C_VEL
LIN {X 0,Y 424.505,Z 754.902,A -85,B 0,C 180,E1 -9819.531,E2 -9819.531} C_VEL
LIN {X 0,Y 424.853,Z 748.885,A -85,B 0,C 180,E1 -9821.45,E2 -9821.45} C_VEL
LIN {X 0,Y 425.423,Z 741.558,A -85,B 0,C 180,E1 -9823.373,E2 -9823.373} C_VEL
LIN {X 0,Y 426.103,Z 732.714,A -85,B 0,C 180,E1 -9825.302,E2 -9825.302} C_VEL
LIN {X 0,Y 426.989,Z 723.579,A -85,B 0,C 180,E1 -9826.988,E2 -9826.988} C_VEL
LIN {X 0,Y 428.192,Z 711.251,A -85,B 0,C 180,E1 -9828.916,E2 -9828.916} C_VEL
LIN {X 0,Y 429.489,Z 698.766,A -85,B 0,C 180,E1 -9830.599,E2 -9830.599} C_VEL
LIN {X 0,Y 431.041,Z 685.092,A -85,B 0,C 180,E1 -9832.152,E2 -9832.152} C_VEL
LIN {X 0,Y 432.463,Z 671.387,A -85,B 0,C 180,E1 -9833.463,E2 -9833.463} C_VEL
LIN {X 0,Y 434.003,Z 656.418,A -85,B 0,C 180,E1 -9834.645,E2 -9834.645} C_VEL
LIN {X 0,Y 435.267,Z 641.98,A -85,B 0,C 180,E1 -9835.59,E2 -9835.59} C_VEL
LIN {X 0,Y 436.873,Z 621.724,A -85,B 0,C 180,E1 -9836.643,E2 -9836.643} C_VEL
LIN {X 0,Y 437.385,Z 612.153,A -85,B 0,C 180,E1 -9837.072,E2 -9837.072} C_VEL
LIN {X 0,Y 432.814,Z 592.328,A -85,B 0,C 180,E1 -9838.152,E2 -9838.152} C_VEL
LIN {X 0,Y 429.033,Z 573.864,A -85,B 0,C 180,E1 -9838.99,E2 -9838.99} C_VEL
LIN {X 0,Y 427.358,Z 566.478,A -85,B 0,C 180,E1 -9839.356,E2 -9839.356} C_VEL
LIN {X 0,Y 427.813,Z 554.207,A -85,B 0,C 180,E1 -9842.549,E2 -9842.549} C_VEL
LIN {X 0,Y 428.458,Z 541.813,A -85,B 0,C 180,E1 -9845.903,E2 -9845.903} C_VEL
LIN {X 0,Y 429.008,Z 530.84,A -85,B 0,C 180,E1 -9849.094,E2 -9849.094} C_VEL
LIN {X 0,Y 429.237,Z 526.979,A -85,B 0,C 180,E1 -9850.297,E2 -9850.297} C_VEL
LIN {X 0,Y 428.454,Z 520.988,A -85,B 0,C 180,E1 -9852.427,E2 -9852.427} C_VEL
LIN {X 0,Y 427.323,Z 514.907,A -85,B 0,C 180,E1 -9855.009,E2 -9855.009} C_VEL
LIN {X 0,Y 426.309,Z 510.425,A -85,B 0,C 180,E1 -9857.475,E2 -9857.475} C_VEL
LIN {X 0,Y 425.647,Z 507.229,A -85,B 0,C 180,E1 -9859.914,E2 -9859.914} C_VEL
LIN {X 0,Y 425.3,Z 505.822,A -85,B 0,C 180,E1 -9861.708,E2 -9861.708} C_VEL
LIN {X 0,Y 425.302,Z 505.822,A -85,B 0,C 180,E1 -9864.665,E2 -9864.665} C_VEL
LIN {X 0,Y 425.266,Z 505.826,A -85,B 0,C 180,E1 -9868.074,E2 -9868.074} C_VEL
LIN {X 0,Y 425.328,Z 505.825,A -85,B 0,C 180,E1 -9871.176,E2 -9871.176} C_VEL
LIN {X 0,Y 426.354,Z 508.7,A -85,B 0,C 180,E1 -9871.371,E2 -9871.371} C_VEL
LIN {X 0,Y 427.678,Z 510.865,A -85,B 0,C 180,E1 -9871.572,E2 -9871.572} C_VEL
LIN {X 0,Y 433.206,Z 522.046,A -85,B 0,C 180,E1 -9872.489,E2 -9872.489} C_VEL
LIN {X 0,Y 437.476,Z 532.99,A -85,B 0,C 180,E1 -9873.332,E2 -9873.332} C_VEL
LIN {X 0,Y 437.811,Z 535.487,A -85,B 0,C 180,E1 -9873.485,E2 -9873.485} C_VEL
LIN {X 0,Y 436.58,Z 552.789,A -85,B 0,C 180,E1 -9874.384,E2 -9874.384} C_VEL
LIN {X 0,Y 435.201,Z 568.884,A -85,B 0,C 180,E1 -9875.429,E2 -9875.429} C_VEL
LIN {X 0,Y 433.855,Z 583.715,A -85,B 0,C 180,E1 -9876.617,E2 -9876.617} C_VEL
LIN {X 0,Y 432.346,Z 598.519,A -85,B 0,C 180,E1 -9878.046,E2 -9878.046} C_VEL
LIN {X 0,Y 430.991,Z 610.959,A -85,B 0,C 180,E1 -9879.477,E2 -9879.477} C_VEL
LIN {X 0,Y 429.835,Z 621.608,A -85,B 0,C 180,E1 -9880.913,E2 -9880.913} C_VEL
LIN {X 0,Y 428.544,Z 632.445,A -85,B 0,C 180,E1 -9882.628,E2 -9882.628} C_VEL
LIN {X 0,Y 427.529,Z 641.179,A -85,B 0,C 180,E1 -9884.262,E2 -9884.262} C_VEL
LIN {X 0,Y 426.615,Z 650.017,A -85,B 0,C 180,E1 -9886.229,E2 -9886.229} C_VEL
LIN {X 0,Y 425.886,Z 657.026,A -85,B 0,C 180,E1 -9888.096,E2 -9888.096} C_VEL
LIN {X 0,Y 425.353,Z 662.818,A -85,B 0,C 180,E1 -9890.01,E2 -9890.01} C_VEL
LIN {X 0,Y 425.028,Z 667.444,A -85,B 0,C 180,E1 -9891.921,E2 -9891.921} C_VEL
LIN {X 0,Y 424.797,Z 670.197,A -85,B 0,C 180,E1 -9893.35,E2 -9893.35} C_VEL
LIN {X 0,Y 424.56,Z 673.015,A -85,B 0,C 180,E1 -9895.253,E2 -9895.253} C_VEL
LIN {X 0,Y 424.451,Z 674.77,A -85,B 0,C 180,E1 -9897.153,E2 -9897.153} C_VEL
LIN {X 0,Y 424.343,Z 675.618,A -85,B 0,C 180,E1 -9899.051,E2 -9899.051} C_VEL
LIN {X 0,Y 424.326,Z 675.481,A -85,B 0,C 180,E1 -9900.949,E2 -9900.949} C_VEL
LIN {X 0,Y 424.449,Z 674.404,A -85,B 0,C 180,E1 -9902.848,E2 -9902.848} C_VEL
LIN {X 0,Y 424.571,Z 673.528,A -85,B 0,C 180,E1 -9903.797,E2 -9903.797} C_VEL
LIN {X 0,Y 424.537,Z 670.98,A -85,B 0,C 180,E1 -9905.701,E2 -9905.701} C_VEL
LIN {X 0,Y 424.791,Z 667.449,A -85,B 0,C 180,E1 -9907.606,E2 -9907.606} C_VEL
LIN {X 0,Y 425.027,Z 662.814,A -85,B 0,C 180,E1 -9909.518,E2 -9909.518} C_VEL
LIN {X 0,Y 425.4,Z 657.024,A -85,B 0,C 180,E1 -9911.435,E2 -9911.435} C_VEL
LIN {X 0,Y 426.114,Z 649.972,A -85,B 0,C 180,E1 -9913.351,E2 -9913.351} C_VEL
LIN {X 0,Y 426.879,Z 641.438,A -85,B 0,C 180,E1 -9915.273,E2 -9915.273} C_VEL
LIN {X 0,Y 427.941,Z 631.209,A -85,B 0,C 180,E1 -9917.195,E2 -9917.195} C_VEL
LIN {X 0,Y 429.054,Z 620.619,A -85,B 0,C 180,E1 -9918.876,E2 -9918.876} C_VEL
LIN {X 0,Y 430.421,Z 608.153,A -85,B 0,C 180,E1 -9920.552,E2 -9920.552} C_VEL
LIN {X 0,Y 431.743,Z 595.594,A -85,B 0,C 180,E1 -9921.988,E2 -9921.988} C_VEL
LIN {X 0,Y 433.152,Z 582.038,A -85,B 0,C 180,E1 -9923.297,E2 -9923.297} C_VEL
LIN {X 0,Y 434.435,Z 568.858,A -85,B 0,C 180,E1 -9924.364,E2 -9924.364} C_VEL
LIN {X 0,Y 435.567,Z 554.286,A -85,B 0,C 180,E1 -9925.367,E2 -9925.367} C_VEL
LIN {X 0,Y 436.781,Z 538.968,A -85,B 0,C 180,E1 -9926.22,E2 -9926.22} C_VEL
LIN {X 0,Y 437.079,Z 534.084,A -85,B 0,C 180,E1 -9926.452,E2 -9926.452} C_VEL
LIN {X 0,Y 431.372,Z 519.79,A -85,B 0,C 180,E1 -9927.451,E2 -9927.451} C_VEL
LIN {X 0,Y 425.491,Z 506.65,A -85,B 0,C 180,E1 -9928.303,E2 -9928.303} C_VEL
LIN {X 0,Y 425.355,Z 505.812,A -85,B 0,C 180,E1 -9928.345,E2 -9928.345} C_VEL
LIN {X 0,Y 425.27,Z 505.827,A -85,B 0,C 180,E1 -9931.927,E2 -9931.927} C_VEL
LIN {X 0,Y 425.305,Z 505.82,A -85,B 0,C 180,E1 -9935.336,E2 -9935.336} C_VEL
LIN {X 0,Y 425.314,Z 505.821,A -85,B 0,C 180,E1 -9938.898,E2 -9938.898} C_VEL
LIN {X 0,Y 425.295,Z 505.823,A -85,B 0,C 180,E1 -9941.958,E2 -9941.958} C_VEL
LIN {X 0,Y 425.29,Z 505.821,A -85,B 0,C 180,E1 -9945.283,E2 -9945.283} C_VEL
LIN {X 0,Y 425.281,Z 505.824,A -85,B 0,C 180,E1 -9948.621,E2 -9948.621} C_VEL
LIN {X 0,Y 425.318,Z 505.819,A -85,B 0,C 180,E1 -9951.103,E2 -9951.103} C_VEL
LIN {X 0,Y 425.305,Z 505.823,A -85,B 0,C 180,E1 -9954.664,E2 -9954.664} C_VEL
LIN {X 0,Y 425.271,Z 505.83,A -85,B 0,C 180,E1 -9958.073,E2 -9958.073} C_VEL
LIN {X 0,Y 425.337,Z 505.82,A -85,B 0,C 180,E1 -9961.368,E2 -9961.368} C_VEL
LIN {X 0,Y 425.409,Z 505.909,A -85,B 0,C 180,E1 -9963.64,E2 -9963.64} C_VEL
LIN {X 0,Y 425.783,Z 509.309,A -85,B 0,C 180,E1 -9965.628,E2 -9965.628} C_VEL
LIN {X 0,Y 425.737,Z 514.608,A -85,B 0,C 180,E1 -9968.704,E2 -9968.704} C_VEL
LIN {X 0,Y 425.685,Z 519.733,A -85,B 0,C 180,E1 -9971.718,E2 -9971.718} C_VEL
LIN {X 0,Y 425.574,Z 524.675,A -85,B 0,C 180,E1 -9974.678,E2 -9974.678} C_VEL
LIN {X 0,Y 425.52,Z 527.029,A -85,B 0,C 180,E1 -9976.094,E2 -9976.094} C_VEL
LIN {X 0,Y 427.41,Z 532.131,A -85,B 0,C 180,E1 -9976.326,E2 -9976.326} C_VEL
LIN {X 0,Y 433.927,Z 548.708,A -85,B 0,C 180,E1 -9977.182,E2 -9977.182} C_VEL
LIN {X 0,Y 438.376,Z 562.011,A -85,B 0,C 180,E1 -9977.947,E2 -9977.947} C_VEL
LIN {X 0,Y 437.354,Z 579.058,A -85,B 0,C 180,E1 -9978.691,E2 -9978.691} C_VEL
LIN {X 0,Y 436.167,Z 594.306,A -85,B 0,C 180,E1 -9979.555,E2 -9979.555} C_VEL
LIN {X 0,Y 435.669,Z 600.092,A -85,B 0,C 180,E1 -9979.937,E2 -9979.937} C_VEL
LIN {X 0,Y 434.52,Z 605.436,A -85,B 0,C 180,E1 -9980.268,E2 -9980.268} C_VEL
LIN {X 0,Y 428.106,Z 620.594,A -85,B 0,C 180,E1 -9981.2,E2 -9981.2} C_VEL
LIN {X 0,Y 426.638,Z 625.372,A -85,B 0,C 180,E1 -9981.593,E2 -9981.593} C_VEL
LIN {X 0,Y 426.396,Z 626.947,A -85,B 0,C 180,E1 -9981.74,E2 -9981.74} C_VEL
LIN {X 0,Y 424.893,Z 639.771,A -85,B 0,C 180,E1 -9983.112,E2 -9983.112} C_VEL
LIN {X 0,Y 423.232,Z 652.79,A -85,B 0,C 180,E1 -9984.759,E2 -9984.759} C_VEL
LIN {X 0,Y 421.856,Z 663.842,A -85,B 0,C 180,E1 -9986.417,E2 -9986.417} C_VEL
LIN {X 0,Y 420.492,Z 674.553,A -85,B 0,C 180,E1 -9988.323,E2 -9988.323} C_VEL
LIN {X 0,Y 419.413,Z 683.556,A -85,B 0,C 180,E1 -9990.239,E2 -9990.239} C_VEL
LIN {X 0,Y 418.664,Z 690.21,A -85,B 0,C 180,E1 -9991.923,E2 -9991.923} C_VEL
LIN {X 0,Y 418.05,Z 696.686,A -85,B 0,C 180,E1 -9993.855,E2 -9993.855} C_VEL
LIN {X 0,Y 417.626,Z 701.911,A -85,B 0,C 180,E1 -9995.794,E2 -9995.794} C_VEL
LIN {X 0,Y 417.366,Z 706.109,A -85,B 0,C 180,E1 -9997.741,E2 -9997.741} C_VEL
LIN {X 0,Y 417.13,Z 709.288,A -85,B 0,C 180,E1 -9999.699,E2 -9999.699} C_VEL
LIN {X 0,Y 417.07,Z 711.887,A -85,B 0,C 180,E1 -10002.215,E2 -10002.215} C_VEL
LIN {X 0,Y 416.957,Z 712.679,A -85,B 0,C 180,E1 -10003.648,E2 -10003.648} C_VEL
LIN {X 0,Y 416.962,Z 712.794,A -85,B 0,C 180,E1 -10006.105,E2 -10006.105} C_VEL
LIN {X 0,Y 416.944,Z 712.124,A -85,B 0,C 180,E1 -10007.661,E2 -10007.661} C_VEL
LIN {X 0,Y 417.039,Z 710.261,A -85,B 0,C 180,E1 -10009.695,E2 -10009.695} C_VEL
LIN {X 0,Y 417.352,Z 706.632,A -85,B 0,C 180,E1 -10012.153,E2 -10012.153} C_VEL
LIN {X 0,Y 417.667,Z 702.239,A -85,B 0,C 180,E1 -10014.261,E2 -10014.261} C_VEL
LIN {X 0,Y 418.217,Z 696.36,A -85,B 0,C 180,E1 -10016.443,E2 -10016.443} C_VEL
LIN {X 0,Y 418.925,Z 689.201,A -85,B 0,C 180,E1 -10018.561,E2 -10018.561} C_VEL
LIN {X 0,Y 419.967,Z 680.363,A -85,B 0,C 180,E1 -10020.689,E2 -10020.689} C_VEL
LIN {X 0,Y 421.113,Z 671.031,A -85,B 0,C 180,E1 -10022.561,E2 -10022.561} C_VEL
LIN {X 0,Y 422.587,Z 659.941,A -85,B 0,C 180,E1 -10024.432,E2 -10024.432} C_VEL
LIN {X 0,Y 424.155,Z 647.974,A -85,B 0,C 180,E1 -10026.131,E2 -10026.131} C_VEL
LIN {X 0,Y 425.761,Z 635.803,A -85,B 0,C 180,E1 -10027.595,E2 -10027.595} C_VEL
LIN {X 0,Y 427.386,Z 622.772,A -85,B 0,C 180,E1 -10028.915,E2 -10028.915} C_VEL
LIN {X 0,Y 428.794,Z 609.675,A -85,B 0,C 180,E1 -10030.037,E2 -10030.037} C_VEL
LIN {X 0,Y 430.311,Z 594.431,A -85,B 0,C 180,E1 -10031.119,E2 -10031.119} C_VEL
LIN {X 0,Y 431.601,Z 579.873,A -85,B 0,C 180,E1 -10031.955,E2 -10031.955} C_VEL
LIN {X 0,Y 432.545,Z 564.054,A -85,B 0,C 180,E1 -10032.673,E2 -10032.673} C_VEL
LIN {X 0,Y 427.613,Z 549.259,A -85,B 0,C 180,E1 -10033.617,E2 -10033.617} C_VEL
LIN {X 0,Y 421.784,Z 535.187,A -85,B 0,C 180,E1 -10034.477,E2 -10034.477} C_VEL
LIN {X 0,Y 418.811,Z 528.64,A -85,B 0,C 180,E1 -10034.866,E2 -10034.866} C_VEL
LIN {X 0,Y 418.734,Z 528.131,A -85,B 0,C 180,E1 -10034.925,E2 -10034.925} C_VEL
LIN {X 0,Y 418.9,Z 523.396,A -85,B 0,C 180,E1 -10037.848,E2 -10037.848} C_VEL
LIN {X 0,Y 418.987,Z 519.11,A -85,B 0,C 180,E1 -10040.495,E2 -10040.495} C_VEL
LIN {X 0,Y 419.118,Z 514.14,A -85,B 0,C 180,E1 -10043.597,E2 -10043.597} C_VEL
LIN {X 0,Y 419.012,Z 511.241,A -85,B 0,C 180,E1 -10045.269,E2 -10045.269} C_VEL
LIN {X 0,Y 418.25,Z 506.743,A -85,B 0,C 180,E1 -10048.076,E2 -10048.076} C_VEL
LIN {X 0,Y 418.269,Z 506.7,A -85,B 0,C 180,E1 -10050.892,E2 -10050.892} C_VEL
LIN {X 0,Y 418.265,Z 506.699,A -85,B 0,C 180,E1 -10054.095,E2 -10054.095} C_VEL
LIN {X 0,Y 418.23,Z 506.702,A -85,B 0,C 180,E1 -10057.263,E2 -10057.263} C_VEL
LIN {X 0,Y 418.307,Z 506.693,A -85,B 0,C 180,E1 -10060.365,E2 -10060.365} C_VEL
LIN {X 0,Y 418.307,Z 506.688,A -85,B 0,C 180,E1 -10063.404,E2 -10063.404} C_VEL
LIN {X 0,Y 418.345,Z 506.686,A -85,B 0,C 180,E1 -10066.993,E2 -10066.993} C_VEL
LIN {X 0,Y 418.35,Z 506.687,A -85,B 0,C 180,E1 -10070.328,E2 -10070.328} C_VEL
LIN {X 0,Y 418.486,Z 506.67,A -85,B 0,C 180,E1 -10073.248,E2 -10073.248} C_VEL
LIN {X 0,Y 418.337,Z 506.683,A -85,B 0,C 180,E1 -10075.181,E2 -10075.181} C_VEL
LIN {X 0,Y 418.535,Z 506.658,A -85,B 0,C 180,E1 -10078.075,E2 -10078.075} C_VEL
LIN {X 0,Y 418.663,Z 506.648,A -85,B 0,C 180,E1 -10080,E2 -10080} C_VEL
LIN {X 0,Y 418.502,Z 506.665,A -85,B 0,C 180,E1 -10082.887,E2 -10082.887} C_VEL
LIN {X 0,Y 418.482,Z 506.668,A -85,B 0,C 180,E1 -10086.751,E2 -10086.751} C_VEL
LIN {X 0,Y 418.35,Z 506.681,A -85,B 0,C 180,E1 -10089.671,E2 -10089.671} C_VEL
LIN {X 0,Y 418.344,Z 506.681,A -85,B 0,C 180,E1 -10093.007,E2 -10093.007} C_VEL
LIN {X 0,Y 418.301,Z 506.666,A -85,B 0,C 180,E1 -10096.736,E2 -10096.736} C_VEL
LIN {X 0,Y 418.291,Z 506.686,A -85,B 0,C 180,E1 -10099.803,E2 -10099.803} C_VEL
LIN {X 0,Y 418.276,Z 506.687,A -85,B 0,C 180,E1 -10102.734,E2 -10102.734} C_VEL
LIN {X 0,Y 418.262,Z 506.681,A -85,B 0,C 180,E1 -10105.904,E2 -10105.904} C_VEL
LIN {X 0,Y 418.264,Z 506.7,A -85,B 0,C 180,E1 -10109.162,E2 -10109.162} C_VEL
LIN {X 0,Y 418.249,Z 506.699,A -85,B 0,C 180,E1 -10112.845,E2 -10112.845} C_VEL
LIN {X 0,Y 418.239,Z 506.698,A -85,B 0,C 180,E1 -10116.239,E2 -10116.239} C_VEL
LIN {X 0,Y 418.29,Z 506.796,A -85,B 0,C 180,E1 -10119.234,E2 -10119.234} C_VEL
LIN {X 0,Y 419.919,Z 514.127,A -85,B 0,C 180,E1 -10122.025,E2 -10122.025} C_VEL
LIN {X 0,Y 421.718,Z 522.434,A -85,B 0,C 180,E1 -10125.044,E2 -10125.044} C_VEL
LIN {X 0,Y 423.293,Z 529.855,A -85,B 0,C 180,E1 -10127.631,E2 -10127.631} C_VEL
LIN {X 0,Y 423.898,Z 534.238,A -85,B 0,C 180,E1 -10129.091,E2 -10129.091} C_VEL
LIN {X 0,Y 423.355,Z 542.667,A -85,B 0,C 180,E1 -10131.682,E2 -10131.682} C_VEL
LIN {X 0,Y 422.501,Z 552.432,A -85,B 0,C 180,E1 -10134.595,E2 -10134.595} C_VEL
LIN {X 0,Y 421.828,Z 561.395,A -85,B 0,C 180,E1 -10137.217,E2 -10137.217} C_VEL
LIN {X 0,Y 421.035,Z 572.606,A -85,B 0,C 180,E1 -10140.398,E2 -10140.398} C_VEL
LIN {X 0,Y 426.958,Z 594.724,A -85,B 0,C 180,E1 -10141.394,E2 -10141.394} C_VEL
LIN {X 0,Y 431.268,Z 612.828,A -85,B 0,C 180,E1 -10142.355,E2 -10142.355} C_VEL
LIN {X 0,Y 431.548,Z 616.079,A -85,B 0,C 180,E1 -10142.521,E2 -10142.521} C_VEL
LIN {X 0,Y 430.205,Z 632.754,A -85,B 0,C 180,E1 -10143.306,E2 -10143.306} C_VEL
LIN {X 0,Y 428.634,Z 648.964,A -85,B 0,C 180,E1 -10144.277,E2 -10144.277} C_VEL
LIN {X 0,Y 426.991,Z 664.663,A -85,B 0,C 180,E1 -10145.444,E2 -10145.444} C_VEL
LIN {X 0,Y 425.43,Z 678.139,A -85,B 0,C 180,E1 -10146.643,E2 -10146.643} C_VEL
LIN {X 0,Y 423.85,Z 691.739,A -85,B 0,C 180,E1 -10148.085,E2 -10148.085} C_VEL
LIN {X 0,Y 422.446,Z 703.572,A -85,B 0,C 180,E1 -10149.553,E2 -10149.553} C_VEL
LIN {X 0,Y 421.041,Z 715.348,A -85,B 0,C 180,E1 -10151.259,E2 -10151.259} C_VEL
LIN {X 0,Y 419.978,Z 725.452,A -85,B 0,C 180,E1 -10152.973,E2 -10152.973} C_VEL
LIN {X 0,Y 418.925,Z 735.211,A -85,B 0,C 180,E1 -10154.929,E2 -10154.929} C_VEL
LIN {X 0,Y 418.205,Z 744.15,A -85,B 0,C 180,E1 -10157.082,E2 -10157.082} C_VEL
LIN {X 0,Y 417.59,Z 751.735,A -85,B 0,C 180,E1 -10159.333,E2 -10159.333} C_VEL
LIN {X 0,Y 417.321,Z 757.025,A -85,B 0,C 180,E1 -10161.283,E2 -10161.283} C_VEL
LIN {X 0,Y 417.209,Z 761.138,A -85,B 0,C 180,E1 -10163.229,E2 -10163.229} C_VEL
LIN {X 0,Y 417.069,Z 764.173,A -85,B 0,C 180,E1 -10165.168,E2 -10165.168} C_VEL
LIN {X 0,Y 417.057,Z 766.17,A -85,B 0,C 180,E1 -10167.103,E2 -10167.103} C_VEL
LIN {X 0,Y 417.049,Z 767.141,A -85,B 0,C 180,E1 -10169.035,E2 -10169.035} C_VEL
LIN {X 0,Y 417.049,Z 767.124,A -85,B 0,C 180,E1 -10170.967,E2 -10170.967} C_VEL
LIN {X 0,Y 417.069,Z 766.057,A -85,B 0,C 180,E1 -10172.899,E2 -10172.899} C_VEL
LIN {X 0,Y 417.076,Z 763.992,A -85,B 0,C 180,E1 -10174.834,E2 -10174.834} C_VEL
LIN {X 0,Y 417.212,Z 760.845,A -85,B 0,C 180,E1 -10176.773,E2 -10176.773} C_VEL
LIN {X 0,Y 417.337,Z 756.594,A -85,B 0,C 180,E1 -10178.718,E2 -10178.718} C_VEL
LIN {X 0,Y 417.592,Z 751.133,A -85,B 0,C 180,E1 -10180.67,E2 -10180.67} C_VEL
LIN {X 0,Y 418.097,Z 744.439,A -85,B 0,C 180,E1 -10182.623,E2 -10182.623} C_VEL
LIN {X 0,Y 418.735,Z 736.317,A -85,B 0,C 180,E1 -10184.582,E2 -10184.582} C_VEL
LIN {X 0,Y 419.921,Z 724.091,A -85,B 0,C 180,E1 -10187.032,E2 -10187.032} C_VEL
LIN {X 0,Y 421.171,Z 712.386,A -85,B 0,C 180,E1 -10188.99,E2 -10188.99} C_VEL
LIN {X 0,Y 422.51,Z 700.265,A -85,B 0,C 180,E1 -10190.701,E2 -10190.701} C_VEL
LIN {X 0,Y 424.121,Z 686.97,A -85,B 0,C 180,E1 -10192.27,E2 -10192.27} C_VEL
LIN {X 0,Y 425.584,Z 673.56,A -85,B 0,C 180,E1 -10193.608,E2 -10193.608} C_VEL
LIN {X 0,Y 427.149,Z 659.203,A -85,B 0,C 180,E1 -10194.805,E2 -10194.805} C_VEL
LIN {X 0,Y 428.487,Z 645.497,A -85,B 0,C 180,E1 -10195.763,E2 -10195.763} C_VEL
LIN {X 0,Y 429.762,Z 630.753,A -85,B 0,C 180,E1 -10196.595,E2 -10196.595} C_VEL
LIN {X 0,Y 430.909,Z 613.822,A -85,B 0,C 180,E1 -10197.396,E2 -10197.396} C_VEL
LIN {X 0,Y 426.6,Z 594.113,A -85,B 0,C 180,E1 -10198.54,E2 -10198.54} C_VEL
LIN {X 0,Y 423.068,Z 576.037,A -85,B 0,C 180,E1 -10199.425,E2 -10199.425} C_VEL
LIN {X 0,Y 420.412,Z 564.994,A -85,B 0,C 180,E1 -10199.99,E2 -10199.99} C_VEL
LIN {X 0,Y 420.985,Z 552.159,A -85,B 0,C 180,E1 -10203.43,E2 -10203.43} C_VEL
LIN {X 0,Y 421.556,Z 541.995,A -85,B 0,C 180,E1 -10206.28,E2 -10206.28} C_VEL
LIN {X 0,Y 422.227,Z 530.863,A -85,B 0,C 180,E1 -10209.643,E2 -10209.643} C_VEL
LIN {X 0,Y 422.266,Z 526.93,A -85,B 0,C 180,E1 -10210.955,E2 -10210.955} C_VEL
LIN {X 0,Y 421.134,Z 520.088,A -85,B 0,C 180,E1 -10213.634,E2 -10213.634} C_VEL
LIN {X 0,Y 420.168,Z 515.192,A -85,B 0,C 180,E1 -10215.993,E2 -10215.993} C_VEL
LIN {X 0,Y 419.444,Z 512.042,A -85,B 0,C 180,E1 -10217.916,E2 -10217.916} C_VEL
LIN {X 0,Y 418.751,Z 508.906,A -85,B 0,C 180,E1 -10220.537,E2 -10220.537} C_VEL
LIN {X 0,Y 418.328,Z 507.226,A -85,B 0,C 180,E1 -10222.786,E2 -10222.786} C_VEL
LIN {X 0,Y 418.247,Z 506.7,A -85,B 0,C 180,E1 -10223.977,E2 -10223.977} C_VEL
LIN {X 0,Y 418.259,Z 506.7,A -85,B 0,C 180,E1 -10227.157,E2 -10227.157} C_VEL
LIN {X 0,Y 418.259,Z 506.699,A -85,B 0,C 180,E1 -10230.46,E2 -10230.46} C_VEL
LIN {X 0,Y 419.347,Z 509.677,A -85,B 0,C 180,E1 -10230.699,E2 -10230.699} C_VEL
LIN {X 0,Y 420.67,Z 511.69,A -85,B 0,C 180,E1 -10230.911,E2 -10230.911} C_VEL
LIN {X 0,Y 426.525,Z 523.088,A -85,B 0,C 180,E1 -10231.939,E2 -10231.939} C_VEL
LIN {X 0,Y 430.834,Z 533.837,A -85,B 0,C 180,E1 -10232.823,E2 -10232.823} C_VEL
LIN {X 0,Y 431.445,Z 535.659,A -85,B 0,C 180,E1 -10232.973,E2 -10232.973} C_VEL
LIN {X 0,Y 431.494,Z 539.049,A -85,B 0,C 180,E1 -10233.157,E2 -10233.157} C_VEL
LIN {X 0,Y 430.24,Z 555.254,A -85,B 0,C 180,E1 -10234.04,E2 -10234.04} C_VEL
LIN {X 0,Y 428.856,Z 570.152,A -85,B 0,C 180,E1 -10235.04,E2 -10235.04} C_VEL
LIN {X 0,Y 427.442,Z 584.861,A -85,B 0,C 180,E1 -10236.245,E2 -10236.245} C_VEL
LIN {X 0,Y 425.985,Z 598.478,A -85,B 0,C 180,E1 -10237.573,E2 -10237.573} C_VEL
LIN {X 0,Y 424.625,Z 610.07,A -85,B 0,C 180,E1 -10238.901,E2 -10238.901} C_VEL
LIN {X 0,Y 423.204,Z 622.602,A -85,B 0,C 180,E1 -10240.602,E2 -10240.602} C_VEL
LIN {X 0,Y 421.825,Z 633.406,A -85,B 0,C 180,E1 -10242.347,E2 -10242.347} C_VEL
LIN {X 0,Y 420.587,Z 643.293,A -85,B 0,C 180,E1 -10244.245,E2 -10244.245} C_VEL
LIN {X 0,Y 419.659,Z 651.921,A -85,B 0,C 180,E1 -10246.246,E2 -10246.246} C_VEL
LIN {X 0,Y 418.814,Z 659.45,A -85,B 0,C 180,E1 -10248.383,E2 -10248.383} C_VEL
LIN {X 0,Y 418.339,Z 664.993,A -85,B 0,C 180,E1 -10250.329,E2 -10250.329} C_VEL
LIN {X 0,Y 417.966,Z 669.325,A -85,B 0,C 180,E1 -10252.27,E2 -10252.27} C_VEL
LIN {X 0,Y 417.735,Z 672.589,A -85,B 0,C 180,E1 -10254.207,E2 -10254.207} C_VEL
LIN {X 0,Y 417.551,Z 674.867,A -85,B 0,C 180,E1 -10256.14,E2 -10256.14} C_VEL
LIN {X 0,Y 417.356,Z 676.132,A -85,B 0,C 180,E1 -10258.07,E2 -10258.07} C_VEL
LIN {X 0,Y 417.263,Z 676.505,A -85,B 0,C 180,E1 -10260,E2 -10260} C_VEL
LIN {X 0,Y 417.325,Z 675.836,A -85,B 0,C 180,E1 -10261.931,E2 -10261.931} C_VEL
LIN {X 0,Y 417.539,Z 674.286,A -85,B 0,C 180,E1 -10263.861,E2 -10263.861} C_VEL
LIN {X 0,Y 417.496,Z 671.701,A -85,B 0,C 180,E1 -10265.797,E2 -10265.797} C_VEL
LIN {X 0,Y 417.774,Z 668.138,A -85,B 0,C 180,E1 -10267.735,E2 -10267.735} C_VEL
LIN {X 0,Y 418.029,Z 663.462,A -85,B 0,C 180,E1 -10269.679,E2 -10269.679} C_VEL
LIN {X 0,Y 418.438,Z 657.621,A -85,B 0,C 180,E1 -10271.628,E2 -10271.628} C_VEL
LIN {X 0,Y 419.172,Z 650.521,A -85,B 0,C 180,E1 -10273.576,E2 -10273.576} C_VEL
LIN {X 0,Y 420.013,Z 641.937,A -85,B 0,C 180,E1 -10275.529,E2 -10275.529} C_VEL
LIN {X 0,Y 421.133,Z 631.643,A -85,B 0,C 180,E1 -10277.481,E2 -10277.481} C_VEL
LIN {X 0,Y 422.283,Z 620.971,A -85,B 0,C 180,E1 -10279.19,E2 -10279.19} C_VEL
LIN {X 0,Y 423.731,Z 608.409,A -85,B 0,C 180,E1 -10280.892,E2 -10280.892} C_VEL
LIN {X 0,Y 425.125,Z 595.742,A -85,B 0,C 180,E1 -10282.348,E2 -10282.348} C_VEL
LIN {X 0,Y 426.587,Z 582.093,A -85,B 0,C 180,E1 -10283.677,E2 -10283.677} C_VEL
LIN {X 0,Y 427.934,Z 568.796,A -85,B 0,C 180,E1 -10284.759,E2 -10284.759} C_VEL
LIN {X 0,Y 429,Z 555.207,A -85,B 0,C 180,E1 -10285.706,E2 -10285.706} C_VEL
LIN {X 0,Y 430.322,Z 539.415,A -85,B 0,C 180,E1 -10286.597,E2 -10286.597} C_VEL
LIN {X 0,Y 430.497,Z 536.228,A -85,B 0,C 180,E1 -10286.752,E2 -10286.752} C_VEL
LIN {X 0,Y 426.199,Z 525.117,A -85,B 0,C 180,E1 -10287.567,E2 -10287.567} C_VEL
LIN {X 0,Y 419.279,Z 509.488,A -85,B 0,C 180,E1 -10288.633,E2 -10288.633} C_VEL
LIN {X 0,Y 418.295,Z 506.695,A -85,B 0,C 180,E1 -10288.801,E2 -10288.801} C_VEL
LIN {X 0,Y 418.25,Z 506.7,A -85,B 0,C 180,E1 -10292.528,E2 -10292.528} C_VEL
LIN {X 0,Y 418.265,Z 506.699,A -85,B 0,C 180,E1 -10294.841,E2 -10294.841} C_VEL
LIN {X 0,Y 418.262,Z 506.697,A -85,B 0,C 180,E1 -10298.441,E2 -10298.441} C_VEL
LIN {X 0,Y 418.245,Z 506.7,A -85,B 0,C 180,E1 -10302.233,E2 -10302.233} C_VEL
LIN {X 0,Y 418.241,Z 506.7,A -85,B 0,C 180,E1 -10305.109,E2 -10305.109} C_VEL
LIN {X 0,Y 418.245,Z 506.7,A -85,B 0,C 180,E1 -10307.767,E2 -10307.767} C_VEL
LIN {X 0,Y 418.264,Z 506.699,A -85,B 0,C 180,E1 -10310.618,E2 -10310.618} C_VEL
LIN {X 0,Y 418.249,Z 506.702,A -85,B 0,C 180,E1 -10313.976,E2 -10313.976} C_VEL
LIN {X 0,Y 418.263,Z 506.701,A -85,B 0,C 180,E1 -10317.156,E2 -10317.156} C_VEL
LIN {X 0,Y 418.275,Z 506.699,A -85,B 0,C 180,E1 -10320.895,E2 -10320.895} C_VEL
LIN {X 0,Y 418.366,Z 506.86,A -85,B 0,C 180,E1 -10323.431,E2 -10323.431} C_VEL
LIN {X 0,Y 418.791,Z 509.854,A -85,B 0,C 180,E1 -10325.194,E2 -10325.194} C_VEL
LIN {X 0,Y 418.778,Z 515.242,A -85,B 0,C 180,E1 -10328.332,E2 -10328.332} C_VEL
LIN {X 0,Y 418.676,Z 520.407,A -85,B 0,C 180,E1 -10331.4,E2 -10331.4} C_VEL
LIN {X 0,Y 418.598,Z 525.455,A -85,B 0,C 180,E1 -10334.416,E2 -10334.416} C_VEL
LIN {X 0,Y 418.552,Z 527.463,A -85,B 0,C 180,E1 -10335.611,E2 -10335.611} C_VEL
LIN {X 0,Y 420.563,Z 532.886,A -85,B 0,C 180,E1 -10335.858,E2 -10335.858} C_VEL
LIN {X 0,Y 426.437,Z 547.63,A -85,B 0,C 180,E1 -10336.639,E2 -10336.639} C_VEL
LIN {X 0,Y 431.817,Z 563.247,A -85,B 0,C 180,E1 -10337.563,E2 -10337.563} C_VEL
LIN {X 0,Y 431.888,Z 565.889,A -85,B 0,C 180,E1 -10337.686,E2 -10337.686} C_VEL
LIN {X 0,Y 430.793,Z 581.661,A -85,B 0,C 180,E1 -10338.411,E2 -10338.411} C_VEL
LIN {X 0,Y 429.572,Z 596.408,A -85,B 0,C 180,E1 -10339.274,E2 -10339.274} C_VEL
LIN {X 0,Y 428.171,Z 610.763,A -85,B 0,C 180,E1 -10340.313,E2 -10340.313} C_VEL
LIN {X 0,Y 426.704,Z 624.161,A -85,B 0,C 180,E1 -10341.475,E2 -10341.475} C_VEL
LIN {X 0,Y 426.396,Z 626.947,A -85,B 0,C 180,E1 -10341.74,E2 -10341.74} C_VEL
LIN {X 0,Y 425.277,Z 631.744,A -85,B 0,C 180,E1 -10342.179,E2 -10342.179} C_VEL
LIN {X 0,Y 421.726,Z 639.493,A -85,B 0,C 180,E1 -10342.864,E2 -10342.864} C_VEL
LIN {X 0,Y 418.067,Z 646.891,A -85,B 0,C 180,E1 -10343.613,E2 -10343.613} C_VEL
LIN {X 0,Y 416.796,Z 651.14,A -85,B 0,C 180,E1 -10344.148,E2 -10344.148} C_VEL
LIN {X 0,Y 415.289,Z 662.775,A -85,B 0,C 180,E1 -10345.875,E2 -10345.875} C_VEL
LIN {X 0,Y 413.817,Z 673.706,A -85,B 0,C 180,E1 -10347.809,E2 -10347.809} C_VEL
LIN {X 0,Y 412.59,Z 682.907,A -85,B 0,C 180,E1 -10349.755,E2 -10349.755} C_VEL
LIN {X 0,Y 411.805,Z 689.77,A -85,B 0,C 180,E1 -10351.466,E2 -10351.466} C_VEL
LIN {X 0,Y 411.103,Z 696.366,A -85,B 0,C 180,E1 -10353.429,E2 -10353.429} C_VEL
LIN {X 0,Y 410.67,Z 701.743,A -85,B 0,C 180,E1 -10355.4,E2 -10355.4} C_VEL
LIN {X 0,Y 410.428,Z 705.087,A -85,B 0,C 180,E1 -10356.883,E2 -10356.883} C_VEL
LIN {X 0,Y 410.143,Z 708.656,A -85,B 0,C 180,E1 -10358.87,E2 -10358.87} C_VEL
LIN {X 0,Y 410.002,Z 711.201,A -85,B 0,C 180,E1 -10360.867,E2 -10360.867} C_VEL
LIN {X 0,Y 409.913,Z 712.761,A -85,B 0,C 180,E1 -10362.877,E2 -10362.877} C_VEL
LIN {X 0,Y 409.847,Z 713.379,A -85,B 0,C 180,E1 -10364.904,E2 -10364.904} C_VEL
LIN {X 0,Y 409.851,Z 712.947,A -85,B 0,C 180,E1 -10366.947,E2 -10366.947} C_VEL
LIN {X 0,Y 409.94,Z 711.565,A -85,B 0,C 180,E1 -10369.009,E2 -10369.009} C_VEL
LIN {X 0,Y 410.099,Z 709.029,A -85,B 0,C 180,E1 -10371.092,E2 -10371.092} C_VEL
LIN {X 0,Y 410.418,Z 705.393,A -85,B 0,C 180,E1 -10373.193,E2 -10373.193} C_VEL
LIN {X 0,Y 410.853,Z 700.562,A -85,B 0,C 180,E1 -10375.317,E2 -10375.317} C_VEL
LIN {X 0,Y 411.494,Z 694.308,A -85,B 0,C 180,E1 -10377.459,E2 -10377.459} C_VEL
LIN {X 0,Y 412.36,Z 686.497,A -85,B 0,C 180,E1 -10379.632,E2 -10379.632} C_VEL
LIN {X 0,Y 413.401,Z 678.339,A -85,B 0,C 180,E1 -10381.516,E2 -10381.516} C_VEL
LIN {X 0,Y 414.759,Z 668.6,A -85,B 0,C 180,E1 -10383.414,E2 -10383.414} C_VEL
LIN {X 0,Y 416.429,Z 656.99,A -85,B 0,C 180,E1 -10385.309,E2 -10385.309} C_VEL
LIN {X 0,Y 418.02,Z 645.092,A -85,B 0,C 180,E1 -10386.943,E2 -10386.943} C_VEL
LIN {X 0,Y 419.795,Z 632.246,A -85,B 0,C 180,E1 -10388.426,E2 -10388.426} C_VEL
LIN {X 0,Y 421.545,Z 618.107,A -85,B 0,C 180,E1 -10389.799,E2 -10389.799} C_VEL
LIN {X 0,Y 423.212,Z 603.258,A -85,B 0,C 180,E1 -10390.99,E2 -10390.99} C_VEL
LIN {X 0,Y 424.574,Z 589.532,A -85,B 0,C 180,E1 -10391.902,E2 -10391.902} C_VEL
LIN {X 0,Y 425.914,Z 573.427,A -85,B 0,C 180,E1 -10392.748,E2 -10392.748} C_VEL
LIN {X 0,Y 426.264,Z 565.742,A -85,B 0,C 180,E1 -10393.092,E2 -10393.092} C_VEL
LIN {X 0,Y 421.191,Z 550.53,A -85,B 0,C 180,E1 -10394.107,E2 -10394.107} C_VEL
LIN {X 0,Y 415.023,Z 535.867,A -85,B 0,C 180,E1 -10395.051,E2 -10395.051} C_VEL
LIN {X 0,Y 411.869,Z 529.107,A -85,B 0,C 180,E1 -10395.475,E2 -10395.475} C_VEL
LIN {X 0,Y 411.795,Z 528.623,A -85,B 0,C 180,E1 -10395.508,E2 -10395.508} C_VEL
LIN {X 0,Y 411.962,Z 523.596,A -85,B 0,C 180,E1 -10398.643,E2 -10398.643} C_VEL
LIN {X 0,Y 412.103,Z 518.019,A -85,B 0,C 180,E1 -10402.124,E2 -10402.124} C_VEL
LIN {X 0,Y 412.106,Z 513.27,A -85,B 0,C 180,E1 -10404.941,E2 -10404.941} C_VEL
LIN {X 0,Y 411.7,Z 510.258,A -85,B 0,C 180,E1 -10406.889,E2 -10406.889} C_VEL
LIN {X 0,Y 411.174,Z 507.587,A -85,B 0,C 180,E1 -10408.715,E2 -10408.715} C_VEL
LIN {X 0,Y 411.216,Z 507.577,A -85,B 0,C 180,E1 -10411.409,E2 -10411.409} C_VEL
LIN {X 0,Y 411.229,Z 507.574,A -85,B 0,C 180,E1 -10414.706,E2 -10414.706} C_VEL
LIN {X 0,Y 411.198,Z 507.58,A -85,B 0,C 180,E1 -10417.913,E2 -10417.913} C_VEL
LIN {X 0,Y 411.226,Z 507.571,A -85,B 0,C 180,E1 -10421.051,E2 -10421.051} C_VEL
LIN {X 0,Y 411.245,Z 507.569,A -85,B 0,C 180,E1 -10424.131,E2 -10424.131} C_VEL
LIN {X 0,Y 411.305,Z 507.565,A -85,B 0,C 180,E1 -10427.165,E2 -10427.165} C_VEL
LIN {X 0,Y 411.299,Z 507.567,A -85,B 0,C 180,E1 -10430.161,E2 -10430.161} C_VEL
LIN {X 0,Y 411.452,Z 507.546,A -85,B 0,C 180,E1 -10433.132,E2 -10433.132} C_VEL
LIN {X 0,Y 411.309,Z 507.558,A -85,B 0,C 180,E1 -10435.099,E2 -10435.099} C_VEL
LIN {X 0,Y 411.504,Z 507.534,A -85,B 0,C 180,E1 -10438.042,E2 -10438.042} C_VEL
LIN {X 0,Y 411.633,Z 507.524,A -85,B 0,C 180,E1 -10440,E2 -10440} C_VEL
LIN {X 0,Y 411.457,Z 507.543,A -85,B 0,C 180,E1 -10442.937,E2 -10442.937} C_VEL
LIN {X 0,Y 411.449,Z 507.544,A -85,B 0,C 180,E1 -10446.867,E2 -10446.867} C_VEL
LIN {X 0,Y 411.298,Z 507.56,A -85,B 0,C 180,E1 -10449.838,E2 -10449.838} C_VEL
LIN {X 0,Y 411.302,Z 507.559,A -85,B 0,C 180,E1 -10453.109,E2 -10453.109} C_VEL
LIN {X 0,Y 411.245,Z 507.542,A -85,B 0,C 180,E1 -10456.889,E2 -10456.889} C_VEL
LIN {X 0,Y 411.244,Z 507.566,A -85,B 0,C 180,E1 -10459.986,E2 -10459.986} C_VEL
LIN {X 0,Y 411.217,Z 507.558,A -85,B 0,C 180,E1 -10463.146,E2 -10463.146} C_VEL
LIN {X 0,Y 411.228,Z 507.564,A -85,B 0,C 180,E1 -10466.381,E2 -10466.381} C_VEL
LIN {X 0,Y 411.2,Z 507.577,A -85,B 0,C 180,E1 -10469.712,E2 -10469.712} C_VEL
LIN {X 0,Y 411.196,Z 507.577,A -85,B 0,C 180,E1 -10473.156,E2 -10473.156} C_VEL
LIN {X 0,Y 411.186,Z 507.576,A -85,B 0,C 180,E1 -10476.554,E2 -10476.554} C_VEL
LIN {X 0,Y 411.234,Z 507.705,A -85,B 0,C 180,E1 -10478.721,E2 -10478.721} C_VEL
LIN {X 0,Y 412.893,Z 515.102,A -85,B 0,C 180,E1 -10481.592,E2 -10481.592} C_VEL
LIN {X 0,Y 414.669,Z 523.274,A -85,B 0,C 180,E1 -10484.618,E2 -10484.618} C_VEL
LIN {X 0,Y 416.627,Z 532.626,A -85,B 0,C 180,E1 -10487.921,E2 -10487.921} C_VEL
LIN {X 0,Y 416.98,Z 536.853,A -85,B 0,C 180,E1 -10489.327,E2 -10489.327} C_VEL
LIN {X 0,Y 416.334,Z 545.376,A -85,B 0,C 180,E1 -10491.967,E2 -10491.967} C_VEL
LIN {X 0,Y 415.461,Z 555.057,A -85,B 0,C 180,E1 -10494.892,E2 -10494.892} C_VEL
LIN {X 0,Y 414.628,Z 565.377,A -85,B 0,C 180,E1 -10497.941,E2 -10497.941} C_VEL
LIN {X 0,Y 414.179,Z 571.939,A -85,B 0,C 180,E1 -10499.847,E2 -10499.847} C_VEL
LIN {X 0,Y 420.368,Z 595.176,A -85,B 0,C 180,E1 -10500.939,E2 -10500.939} C_VEL
LIN {X 0,Y 424.512,Z 613.174,A -85,B 0,C 180,E1 -10501.927,E2 -10501.927} C_VEL
LIN {X 0,Y 425.112,Z 616.505,A -85,B 0,C 180,E1 -10502.121,E2 -10502.121} C_VEL
LIN {X 0,Y 423.698,Z 633.104,A -85,B 0,C 180,E1 -10502.929,E2 -10502.929} C_VEL
LIN {X 0,Y 422.196,Z 647.827,A -85,B 0,C 180,E1 -10503.826,E2 -10503.826} C_VEL
LIN {X 0,Y 420.598,Z 662.465,A -85,B 0,C 180,E1 -10504.914,E2 -10504.914} C_VEL
LIN {X 0,Y 418.949,Z 676.088,A -85,B 0,C 180,E1 -10506.129,E2 -10506.129} C_VEL
LIN {X 0,Y 417.194,Z 690.316,A -85,B 0,C 180,E1 -10507.636,E2 -10507.636} C_VEL
LIN {X 0,Y 415.651,Z 702.818,A -85,B 0,C 180,E1 -10509.203,E2 -10509.203} C_VEL
LIN {X 0,Y 414.169,Z 714.609,A -85,B 0,C 180,E1 -10510.936,E2 -10510.936} C_VEL
LIN {X 0,Y 413.02,Z 724.906,A -85,B 0,C 180,E1 -10512.713,E2 -10512.713} C_VEL
LIN {X 0,Y 411.928,Z 734.481,A -85,B 0,C 180,E1 -10514.667,E2 -10514.667} C_VEL
LIN {X 0,Y 411.193,Z 742.886,A -85,B 0,C 180,E1 -10516.711,E2 -10516.711} C_VEL
LIN {X 0,Y 410.662,Z 749.55,A -85,B 0,C 180,E1 -10518.651,E2 -10518.651} C_VEL
LIN {X 0,Y 410.298,Z 755.094,A -85,B 0,C 180,E1 -10520.636,E2 -10520.636} C_VEL
LIN {X 0,Y 410.171,Z 758.527,A -85,B 0,C 180,E1 -10522.123,E2 -10522.123} C_VEL
LIN {X 0,Y 410.063,Z 762.076,A -85,B 0,C 180,E1 -10524.099,E2 -10524.099} C_VEL
LIN {X 0,Y 409.942,Z 764.612,A -85,B 0,C 180,E1 -10526.069,E2 -10526.069} C_VEL
LIN {X 0,Y 410.062,Z 766.067,A -85,B 0,C 180,E1 -10528.037,E2 -10528.037} C_VEL
LIN {X 0,Y 409.972,Z 766.547,A -85,B 0,C 180,E1 -10530.001,E2 -10530.001} C_VEL
LIN {X 0,Y 410.064,Z 765.973,A -85,B 0,C 180,E1 -10531.965,E2 -10531.965} C_VEL
LIN {X 0,Y 409.979,Z 764.388,A -85,B 0,C 180,E1 -10533.933,E2 -10533.933} C_VEL
LIN {X 0,Y 410.113,Z 761.755,A -85,B 0,C 180,E1 -10535.903,E2 -10535.903} C_VEL
LIN {X 0,Y 410.215,Z 758.032,A -85,B 0,C 180,E1 -10537.879,E2 -10537.879} C_VEL
LIN {X 0,Y 410.362,Z 753.129,A -85,B 0,C 180,E1 -10539.862,E2 -10539.862} C_VEL
LIN {X 0,Y 410.774,Z 747.019,A -85,B 0,C 180,E1 -10541.849,E2 -10541.849} C_VEL
LIN {X 0,Y 411.451,Z 738.721,A -85,B 0,C 180,E1 -10544.088,E2 -10544.088} C_VEL
LIN {X 0,Y 412.356,Z 729.985,A -85,B 0,C 180,E1 -10546.08,E2 -10546.08} C_VEL
LIN {X 0,Y 413.439,Z 719.497,A -85,B 0,C 180,E1 -10548.074,E2 -10548.074} C_VEL
LIN {X 0,Y 414.723,Z 708.642,A -85,B 0,C 180,E1 -10549.812,E2 -10549.812} C_VEL
LIN {X 0,Y 416.008,Z 697.87,A -85,B 0,C 180,E1 -10551.299,E2 -10551.299} C_VEL
LIN {X 0,Y 417.574,Z 685.393,A -85,B 0,C 180,E1 -10552.775,E2 -10552.775} C_VEL
LIN {X 0,Y 419.271,Z 670.522,A -85,B 0,C 180,E1 -10554.248,E2 -10554.248} C_VEL
LIN {X 0,Y 420.845,Z 656.482,A -85,B 0,C 180,E1 -10555.392,E2 -10555.392} C_VEL
LIN {X 0,Y 422.382,Z 641.027,A -85,B 0,C 180,E1 -10556.43,E2 -10556.43} C_VEL
LIN {X 0,Y 423.736,Z 625.326,A -85,B 0,C 180,E1 -10557.271,E2 -10557.271} C_VEL
LIN {X 0,Y 424.449,Z 616.282,A -85,B 0,C 180,E1 -10557.689,E2 -10557.689} C_VEL
LIN {X 0,Y 420.367,Z 595.538,A -85,B 0,C 180,E1 -10558.961,E2 -10558.961} C_VEL
LIN {X 0,Y 417.017,Z 577.529,A -85,B 0,C 180,E1 -10559.905,E2 -10559.905} C_VEL
LIN {X 0,Y 414.163,Z 566.572,A -85,B 0,C 180,E1 -10560.529,E2 -10560.529} C_VEL
LIN {X 0,Y 413.456,Z 563.261,A -85,B 0,C 180,E1 -10560.732,E2 -10560.732} C_VEL
LIN {X 0,Y 414.107,Z 551.222,A -85,B 0,C 180,E1 -10564.061,E2 -10564.061} C_VEL
LIN {X 0,Y 414.672,Z 541.816,A -85,B 0,C 180,E1 -10566.796,E2 -10566.796} C_VEL
LIN {X 0,Y 415.39,Z 531.589,A -85,B 0,C 180,E1 -10570.011,E2 -10570.011} C_VEL
LIN {X 0,Y 415.295,Z 527.933,A -85,B 0,C 180,E1 -10571.3,E2 -10571.3} C_VEL
LIN {X 0,Y 414.316,Z 522.012,A -85,B 0,C 180,E1 -10573.722,E2 -10573.722} C_VEL
LIN {X 0,Y 413.507,Z 517.721,A -85,B 0,C 180,E1 -10575.827,E2 -10575.827} C_VEL
LIN {X 0,Y 412.497,Z 513.45,A -85,B 0,C 180,E1 -10578.562,E2 -10578.562} C_VEL
LIN {X 0,Y 411.955,Z 510.914,A -85,B 0,C 180,E1 -10580.86,E2 -10580.86} C_VEL
LIN {X 0,Y 411.537,Z 509.148,A -85,B 0,C 180,E1 -10583.384,E2 -10583.384} C_VEL
LIN {X 0,Y 411.339,Z 508.304,A -85,B 0,C 180,E1 -10585.68,E2 -10585.68} C_VEL
LIN {X 0,Y 411.262,Z 508.059,A -85,B 0,C 180,E1 -10588.699,E2 -10588.699} C_VEL
LIN {X 0,Y 411.297,Z 508.145,A -85,B 0,C 180,E1 -10589.722,E2 -10589.722} C_VEL
LIN {X 0,Y 412.544,Z 510.899,A -85,B 0,C 180,E1 -10589.991,E2 -10589.991} C_VEL
LIN {X 0,Y 413.702,Z 512.547,A -85,B 0,C 180,E1 -10590.188,E2 -10590.188} C_VEL
LIN {X 0,Y 419.365,Z 523.192,A -85,B 0,C 180,E1 -10591.25,E2 -10591.25} C_VEL
LIN {X 0,Y 424.144,Z 534.415,A -85,B 0,C 180,E1 -10592.256,E2 -10592.256} C_VEL
LIN {X 0,Y 425.515,Z 539.006,A -85,B 0,C 180,E1 -10592.637,E2 -10592.637} C_VEL
LIN {X 0,Y 424.184,Z 555.287,A -85,B 0,C 180,E1 -10593.529,E2 -10593.529} C_VEL
LIN {X 0,Y 422.568,Z 571.559,A -85,B 0,C 180,E1 -10594.643,E2 -10594.643} C_VEL
LIN {X 0,Y 421.074,Z 586.159,A -85,B 0,C 180,E1 -10595.863,E2 -10595.863} C_VEL
LIN {X 0,Y 419.535,Z 599.498,A -85,B 0,C 180,E1 -10597.195,E2 -10597.195} C_VEL
LIN {X 0,Y 418.086,Z 611.204,A -85,B 0,C 180,E1 -10598.555,E2 -10598.555} C_VEL
LIN {X 0,Y 416.565,Z 623.632,A -85,B 0,C 180,E1 -10600.28,E2 -10600.28} C_VEL
LIN {X 0,Y 415.109,Z 634.451,A -85,B 0,C 180,E1 -10602.056,E2 -10602.056} C_VEL
LIN {X 0,Y 413.985,Z 643.101,A -85,B 0,C 180,E1 -10603.734,E2 -10603.734} C_VEL
LIN {X 0,Y 412.904,Z 651.901,A -85,B 0,C 180,E1 -10605.762,E2 -10605.762} C_VEL
LIN {X 0,Y 412.071,Z 658.881,A -85,B 0,C 180,E1 -10607.691,E2 -10607.691} C_VEL
LIN {X 0,Y 411.466,Z 664.637,A -85,B 0,C 180,E1 -10609.669,E2 -10609.669} C_VEL
LIN {X 0,Y 411.105,Z 668.228,A -85,B 0,C 180,E1 -10611.15,E2 -10611.15} C_VEL
LIN {X 0,Y 410.819,Z 671.965,A -85,B 0,C 180,E1 -10613.123,E2 -10613.123} C_VEL
LIN {X 0,Y 410.519,Z 674.753,A -85,B 0,C 180,E1 -10615.09,E2 -10615.09} C_VEL
LIN {X 0,Y 410.379,Z 676.47,A -85,B 0,C 180,E1 -10617.055,E2 -10617.055} C_VEL
LIN {X 0,Y 410.243,Z 677.273,A -85,B 0,C 180,E1 -10619.019,E2 -10619.019} C_VEL
LIN {X 0,Y 410.221,Z 677.09,A -85,B 0,C 180,E1 -10620.982,E2 -10620.982} C_VEL
LIN {X 0,Y 410.376,Z 675.945,A -85,B 0,C 180,E1 -10622.945,E2 -10622.945} C_VEL
LIN {X 0,Y 410.508,Z 675.039,A -85,B 0,C 180,E1 -10623.927,E2 -10623.927} C_VEL
LIN {X 0,Y 410.457,Z 672.424,A -85,B 0,C 180,E1 -10625.897,E2 -10625.897} C_VEL
LIN {X 0,Y 410.746,Z 668.811,A -85,B 0,C 180,E1 -10627.868,E2 -10627.868} C_VEL
LIN {X 0,Y 411.041,Z 664.101,A -85,B 0,C 180,E1 -10629.845,E2 -10629.845} C_VEL
LIN {X 0,Y 411.475,Z 658.198,A -85,B 0,C 180,E1 -10631.828,E2 -10631.828} C_VEL
LIN {X 0,Y 412.235,Z 651.028,A -85,B 0,C 180,E1 -10633.809,E2 -10633.809} C_VEL
LIN {X 0,Y 413.138,Z 642.388,A -85,B 0,C 180,E1 -10635.795,E2 -10635.795} C_VEL
LIN {X 0,Y 414.321,Z 632.007,A -85,B 0,C 180,E1 -10637.778,E2 -10637.778} C_VEL
LIN {X 0,Y 415.527,Z 621.252,A -85,B 0,C 180,E1 -10639.515,E2 -10639.515} C_VEL
LIN {X 0,Y 417.05,Z 608.593,A -85,B 0,C 180,E1 -10641.243,E2 -10641.243} C_VEL
LIN {X 0,Y 418.642,Z 594.642,A -85,B 0,C 180,E1 -10642.844,E2 -10642.844} C_VEL
LIN {X 0,Y 420.147,Z 580.63,A -85,B 0,C 180,E1 -10644.194,E2 -10644.194} C_VEL
LIN {X 0,Y 421.613,Z 567.119,A -85,B 0,C 180,E1 -10645.287,E2 -10645.287} C_VEL
LIN {X 0,Y 422.772,Z 553.16,A -85,B 0,C 180,E1 -10646.234,E2 -10646.234} C_VEL
LIN {X 0,Y 423.889,Z 538.917,A -85,B 0,C 180,E1 -10647.033,E2 -10647.033} C_VEL
LIN {X 0,Y 423.813,Z 537.514,A -85,B 0,C 180,E1 -10647.112,E2 -10647.112} C_VEL
LIN {X 0,Y 417.694,Z 522.513,A -85,B 0,C 180,E1 -10648.252,E2 -10648.252} C_VEL
LIN {X 0,Y 411.399,Z 508.417,A -85,B 0,C 180,E1 -10649.216,E2 -10649.216} C_VEL
LIN {X 0,Y 411.238,Z 507.573,A -85,B 0,C 180,E1 -10649.277,E2 -10649.277} C_VEL
LIN {X 0,Y 411.211,Z 507.578,A -85,B 0,C 180,E1 -10653.156,E2 -10653.156} C_VEL
LIN {X 0,Y 411.2,Z 507.577,A -85,B 0,C 180,E1 -10656.553,E2 -10656.553} C_VEL
LIN {X 0,Y 411.219,Z 507.575,A -85,B 0,C 180,E1 -10659.728,E2 -10659.728} C_VEL
LIN {X 0,Y 411.178,Z 507.582,A -85,B 0,C 180,E1 -10663.134,E2 -10663.134} C_VEL
LIN {X 0,Y 411.173,Z 507.582,A -85,B 0,C 180,E1 -10665.881,E2 -10665.881} C_VEL
LIN {X 0,Y 411.17,Z 507.582,A -85,B 0,C 180,E1 -10668.771,E2 -10668.771} C_VEL
LIN {X 0,Y 411.213,Z 507.579,A -85,B 0,C 180,E1 -10671.831,E2 -10671.831} C_VEL
LIN {X 0,Y 411.217,Z 507.576,A -85,B 0,C 180,E1 -10675.121,E2 -10675.121} C_VEL
LIN {X 0,Y 411.172,Z 507.587,A -85,B 0,C 180,E1 -10678.002,E2 -10678.002} C_VEL
LIN {X 0,Y 411.225,Z 507.578,A -85,B 0,C 180,E1 -10681.41,E2 -10681.41} C_VEL
LIN {X 0,Y 411.302,Z 507.587,A -85,B 0,C 180,E1 -10683.076,E2 -10683.076} C_VEL
LIN {X 0,Y 411.72,Z 510.484,A -85,B 0,C 180,E1 -10684.784,E2 -10684.784} C_VEL
LIN {X 0,Y 411.781,Z 515.844,A -85,B 0,C 180,E1 -10687.945,E2 -10687.945} C_VEL
LIN {X 0,Y 411.703,Z 521.11,A -85,B 0,C 180,E1 -10691.074,E2 -10691.074} C_VEL
LIN {X 0,Y 411.604,Z 526.232,A -85,B 0,C 180,E1 -10694.145,E2 -10694.145} C_VEL
LIN {X 0,Y 411.567,Z 527.811,A -85,B 0,C 180,E1 -10695.095,E2 -10695.095} C_VEL
LIN {X 0,Y 413.791,Z 533.682,A -85,B 0,C 180,E1 -10695.386,E2 -10695.386} C_VEL
LIN {X 0,Y 419.747,Z 548.59,A -85,B 0,C 180,E1 -10696.198,E2 -10696.198} C_VEL
LIN {X 0,Y 425.059,Z 564.088,A -85,B 0,C 180,E1 -10697.143,E2 -10697.143} C_VEL
LIN {X 0,Y 425.555,Z 565.824,A -85,B 0,C 180,E1 -10697.256,E2 -10697.256} C_VEL
LIN {X 0,Y 424.425,Z 581.518,A -85,B 0,C 180,E1 -10697.978,E2 -10697.978} C_VEL
LIN {X 0,Y 423.138,Z 596.593,A -85,B 0,C 180,E1 -10698.866,E2 -10698.866} C_VEL
LIN {X 0,Y 421.662,Z 611.029,A -85,B 0,C 180,E1 -10699.92,E2 -10699.92} C_VEL
LIN {X 0,Y 420.072,Z 625.089,A -85,B 0,C 180,E1 -10701.157,E2 -10701.157} C_VEL
LIN {X 0,Y 418.501,Z 638.085,A -85,B 0,C 180,E1 -10702.521,E2 -10702.521} C_VEL
LIN {X 0,Y 416.884,Z 650.603,A -85,B 0,C 180,E1 -10704.074,E2 -10704.074} C_VEL
LIN {X 0,Y 416.796,Z 651.14,A -85,B 0,C 180,E1 -10704.148,E2 -10704.148} C_VEL
LIN {X 0,Y 415.55,Z 655.381,A -85,B 0,C 180,E1 -10704.704,E2 -10704.704} C_VEL
LIN {X 0,Y 408.988,Z 667.226,A -85,B 0,C 180,E1 -10706.314,E2 -10706.314} C_VEL
LIN {X 0,Y 407.488,Z 670.916,A -85,B 0,C 180,E1 -10706.925,E2 -10706.925} C_VEL
LIN {X 0,Y 407.232,Z 672.079,A -85,B 0,C 180,E1 -10707.142,E2 -10707.142} C_VEL
LIN {X 0,Y 405.981,Z 681.153,A -85,B 0,C 180,E1 -10709.007,E2 -10709.007} C_VEL
LIN {X 0,Y 404.974,Z 689.282,A -85,B 0,C 180,E1 -10710.993,E2 -10710.993} C_VEL
LIN {X 0,Y 404.043,Z 697.543,A -85,B 0,C 180,E1 -10713.489,E2 -10713.489} C_VEL
LIN {X 0,Y 403.593,Z 702.774,A -85,B 0,C 180,E1 -10715.495,E2 -10715.495} C_VEL
LIN {X 0,Y 403.341,Z 706.042,A -85,B 0,C 180,E1 -10717.005,E2 -10717.005} C_VEL
LIN {X 0,Y 403.057,Z 709.453,A -85,B 0,C 180,E1 -10719.028,E2 -10719.028} C_VEL
LIN {X 0,Y 402.933,Z 711.922,A -85,B 0,C 180,E1 -10721.06,E2 -10721.06} C_VEL
LIN {X 0,Y 402.828,Z 713.33,A -85,B 0,C 180,E1 -10723.108,E2 -10723.108} C_VEL
LIN {X 0,Y 402.766,Z 713.843,A -85,B 0,C 180,E1 -10725.172,E2 -10725.172} C_VEL
LIN {X 0,Y 402.774,Z 713.285,A -85,B 0,C 180,E1 -10727.254,E2 -10727.254} C_VEL
LIN {X 0,Y 402.896,Z 711.465,A -85,B 0,C 180,E1 -10729.615,E2 -10729.615} C_VEL
LIN {X 0,Y 403.08,Z 709.126,A -85,B 0,C 180,E1 -10731.477,E2 -10731.477} C_VEL
LIN {X 0,Y 403.444,Z 705.319,A -85,B 0,C 180,E1 -10733.618,E2 -10733.618} C_VEL
LIN {X 0,Y 403.939,Z 700.311,A -85,B 0,C 180,E1 -10735.782,E2 -10735.782} C_VEL
LIN {X 0,Y 404.66,Z 693.947,A -85,B 0,C 180,E1 -10737.963,E2 -10737.963} C_VEL
LIN {X 0,Y 405.615,Z 685.98,A -85,B 0,C 180,E1 -10740.162,E2 -10740.162} C_VEL
LIN {X 0,Y 406.866,Z 677.136,A -85,B 0,C 180,E1 -10742.177,E2 -10742.177} C_VEL
LIN {X 0,Y 408.206,Z 667.921,A -85,B 0,C 180,E1 -10743.956,E2 -10743.956} C_VEL
LIN {X 0,Y 409.811,Z 657.549,A -85,B 0,C 180,E1 -10745.666,E2 -10745.666} C_VEL
LIN {X 0,Y 411.471,Z 645.669,A -85,B 0,C 180,E1 -10747.324,E2 -10747.324} C_VEL
LIN {X 0,Y 413.282,Z 633.269,A -85,B 0,C 180,E1 -10748.782,E2 -10748.782} C_VEL
LIN {X 0,Y 415.09,Z 619.398,A -85,B 0,C 180,E1 -10750.163,E2 -10750.163} C_VEL
LIN {X 0,Y 416.747,Z 605.933,A -85,B 0,C 180,E1 -10751.283,E2 -10751.283} C_VEL
LIN {X 0,Y 418.166,Z 592.021,A -85,B 0,C 180,E1 -10752.24,E2 -10752.24} C_VEL
LIN {X 0,Y 419.469,Z 577.659,A -85,B 0,C 180,E1 -10753.04,E2 -10753.04} C_VEL
LIN {X 0,Y 420.013,Z 567.627,A -85,B 0,C 180,E1 -10753.517,E2 -10753.517} C_VEL
LIN {X 0,Y 415.036,Z 552.478,A -85,B 0,C 180,E1 -10754.574,E2 -10754.574} C_VEL
LIN {X 0,Y 408.887,Z 537.992,A -85,B 0,C 180,E1 -10755.558,E2 -10755.558} C_VEL
LIN {X 0,Y 405.022,Z 529.843,A -85,B 0,C 180,E1 -10756.1,E2 -10756.1} C_VEL
LIN {X 0,Y 404.859,Z 529.066,A -85,B 0,C 180,E1 -10756.168,E2 -10756.168} C_VEL
LIN {X 0,Y 405.017,Z 524.931,A -85,B 0,C 180,E1 -10758.746,E2 -10758.746} C_VEL
LIN {X 0,Y 405.168,Z 519.751,A -85,B 0,C 180,E1 -10761.991,E2 -10761.991} C_VEL
LIN {X 0,Y 405.2,Z 514.712,A -85,B 0,C 180,E1 -10765.084,E2 -10765.084} C_VEL
LIN {X 0,Y 404.655,Z 511.196,A -85,B 0,C 180,E1 -10767.424,E2 -10767.424} C_VEL
LIN {X 0,Y 404.146,Z 508.46,A -85,B 0,C 180,E1 -10769.136,E2 -10769.136} C_VEL
LIN {X 0,Y 404.218,Z 508.449,A -85,B 0,C 180,E1 -10772.46,E2 -10772.46} C_VEL
LIN {X 0,Y 404.169,Z 508.454,A -85,B 0,C 180,E1 -10775.333,E2 -10775.333} C_VEL
LIN {X 0,Y 404.155,Z 508.455,A -85,B 0,C 180,E1 -10778.581,E2 -10778.581} C_VEL
LIN {X 0,Y 404.204,Z 508.449,A -85,B 0,C 180,E1 -10781.761,E2 -10781.761} C_VEL
LIN {X 0,Y 404.198,Z 508.451,A -85,B 0,C 180,E1 -10784.881,E2 -10784.881} C_VEL
LIN {X 0,Y 404.26,Z 508.443,A -85,B 0,C 180,E1 -10787.958,E2 -10787.958} C_VEL
LIN {X 0,Y 404.423,Z 508.415,A -85,B 0,C 180,E1 -10792.099,E2 -10792.099} C_VEL
LIN {X 0,Y 404.429,Z 508.42,A -85,B 0,C 180,E1 -10794.015,E2 -10794.015} C_VEL
LIN {X 0,Y 404.473,Z 508.41,A -85,B 0,C 180,E1 -10798.008,E2 -10798.008} C_VEL
LIN {X 0,Y 404.602,Z 508.4,A -85,B 0,C 180,E1 -10800,E2 -10800} C_VEL
LIN {X 0,Y 404.414,Z 508.42,A -85,B 0,C 180,E1 -10802.988,E2 -10802.988} C_VEL
LIN {X 0,Y 404.4,Z 508.423,A -85,B 0,C 180,E1 -10806.987,E2 -10806.987} C_VEL
LIN {X 0,Y 404.261,Z 508.438,A -85,B 0,C 180,E1 -10810.011,E2 -10810.011} C_VEL
LIN {X 0,Y 404.255,Z 508.437,A -85,B 0,C 180,E1 -10813.211,E2 -10813.211} C_VEL
LIN {X 0,Y 404.204,Z 508.416,A -85,B 0,C 180,E1 -10817.007,E2 -10817.007} C_VEL
LIN {X 0,Y 404.195,Z 508.448,A -85,B 0,C 180,E1 -10820.349,E2 -10820.349} C_VEL
LIN {X 0,Y 404.171,Z 508.427,A -85,B 0,C 180,E1 -10823.574,E2 -10823.574} C_VEL
LIN {X 0,Y 404.185,Z 508.447,A -85,B 0,C 180,E1 -10826.877,E2 -10826.877} C_VEL
LIN {X 0,Y 404.144,Z 508.457,A -85,B 0,C 180,E1 -10830.285,E2 -10830.285} C_VEL
LIN {X 0,Y 404.135,Z 508.457,A -85,B 0,C 180,E1 -10833.813,E2 -10833.813} C_VEL
LIN {X 0,Y 404.131,Z 508.455,A -85,B 0,C 180,E1 -10836.877,E2 -10836.877} C_VEL
LIN {X 0,Y 404.216,Z 508.653,A -85,B 0,C 180,E1 -10838.226,E2 -10838.226} C_VEL
LIN {X 0,Y 405.871,Z 516.039,A -85,B 0,C 180,E1 -10841.147,E2 -10841.147} C_VEL
LIN {X 0,Y 408.042,Z 526.103,A -85,B 0,C 180,E1 -10844.924,E2 -10844.924} C_VEL
LIN {X 0,Y 409.838,Z 534.807,A -85,B 0,C 180,E1 -10848.029,E2 -10848.029} C_VEL
LIN {X 0,Y 410.093,Z 538.837,A -85,B 0,C 180,E1 -10849.368,E2 -10849.368} C_VEL
LIN {X 0,Y 409.306,Z 547.757,A -85,B 0,C 180,E1 -10852.17,E2 -10852.17} C_VEL
LIN {X 0,Y 408.406,Z 558.335,A -85,B 0,C 180,E1 -10855.4,E2 -10855.4} C_VEL
LIN {X 0,Y 407.341,Z 571.398,A -85,B 0,C 180,E1 -10859.289,E2 -10859.289} C_VEL
LIN {X 0,Y 413.677,Z 595.105,A -85,B 0,C 180,E1 -10860.445,E2 -10860.445} C_VEL
LIN {X 0,Y 417.734,Z 613.166,A -85,B 0,C 180,E1 -10861.465,E2 -10861.465} C_VEL
LIN {X 0,Y 418.63,Z 617.619,A -85,B 0,C 180,E1 -10861.737,E2 -10861.737} C_VEL
LIN {X 0,Y 417.135,Z 634.546,A -85,B 0,C 180,E1 -10862.604,E2 -10862.604} C_VEL
LIN {X 0,Y 415.547,Z 648.8,A -85,B 0,C 180,E1 -10863.51,E2 -10863.51} C_VEL
LIN {X 0,Y 413.872,Z 663.316,A -85,B 0,C 180,E1 -10864.628,E2 -10864.628} C_VEL
LIN {X 0,Y 412.03,Z 677.86,A -85,B 0,C 180,E1 -10865.97,E2 -10865.97} C_VEL
LIN {X 0,Y 410.243,Z 691.489,A -85,B 0,C 180,E1 -10867.476,E2 -10867.476} C_VEL
LIN {X 0,Y 408.639,Z 703.866,A -85,B 0,C 180,E1 -10869.093,E2 -10869.093} C_VEL
LIN {X 0,Y 407.133,Z 715.383,A -85,B 0,C 180,E1 -10870.855,E2 -10870.855} C_VEL
LIN {X 0,Y 405.81,Z 726.562,A -85,B 0,C 180,E1 -10872.879,E2 -10872.879} C_VEL
LIN {X 0,Y 404.854,Z 734.896,A -85,B 0,C 180,E1 -10874.65,E2 -10874.65} C_VEL
LIN {X 0,Y 404.168,Z 742.166,A -85,B 0,C 180,E1 -10876.476,E2 -10876.476} C_VEL
LIN {X 0,Y 403.614,Z 748.841,A -85,B 0,C 180,E1 -10878.45,E2 -10878.45} C_VEL
LIN {X 0,Y 403.217,Z 754.383,A -85,B 0,C 180,E1 -10880.47,E2 -10880.47} C_VEL
LIN {X 0,Y 403.108,Z 757.82,A -85,B 0,C 180,E1 -10881.984,E2 -10881.984} C_VEL
LIN {X 0,Y 402.998,Z 761.374,A -85,B 0,C 180,E1 -10883.995,E2 -10883.995} C_VEL
LIN {X 0,Y 402.871,Z 763.902,A -85,B 0,C 180,E1 -10886,E2 -10886} C_VEL
LIN {X 0,Y 403.001,Z 765.351,A -85,B 0,C 180,E1 -10888.002,E2 -10888.002} C_VEL
LIN {X 0,Y 402.926,Z 765.818,A -85,B 0,C 180,E1 -10890.001,E2 -10890.001} C_VEL
LIN {X 0,Y 403.021,Z 765.231,A -85,B 0,C 180,E1 -10892,E2 -10892} C_VEL
LIN {X 0,Y 402.928,Z 763.611,A -85,B 0,C 180,E1 -10894.002,E2 -10894.002} C_VEL
LIN {X 0,Y 403.062,Z 760.961,A -85,B 0,C 180,E1 -10896.006,E2 -10896.006} C_VEL
LIN {X 0,Y 403.144,Z 757.187,A -85,B 0,C 180,E1 -10898.018,E2 -10898.018} C_VEL
LIN {X 0,Y 403.415,Z 750.919,A -85,B 0,C 180,E1 -10900.541,E2 -10900.541} C_VEL
LIN {X 0,Y 403.912,Z 744.773,A -85,B 0,C 180,E1 -10902.563,E2 -10902.563} C_VEL
LIN {X 0,Y 404.544,Z 737.245,A -85,B 0,C 180,E1 -10904.591,E2 -10904.591} C_VEL
LIN {X 0,Y 405.538,Z 728.288,A -85,B 0,C 180,E1 -10906.616,E2 -10906.616} C_VEL
LIN {X 0,Y 406.564,Z 719.052,A -85,B 0,C 180,E1 -10908.39,E2 -10908.39} C_VEL
LIN {X 0,Y 407.928,Z 708.2,A -85,B 0,C 180,E1 -10910.156,E2 -10910.156} C_VEL
LIN {X 0,Y 409.452,Z 696.266,A -85,B 0,C 180,E1 -10911.812,E2 -10911.812} C_VEL
LIN {X 0,Y 411.052,Z 683.746,A -85,B 0,C 180,E1 -10913.291,E2 -10913.291} C_VEL
LIN {X 0,Y 412.711,Z 670.03,A -85,B 0,C 180,E1 -10914.659,E2 -10914.659} C_VEL
LIN {X 0,Y 414.427,Z 655.11,A -85,B 0,C 180,E1 -10915.887,E2 -10915.887} C_VEL
LIN {X 0,Y 415.974,Z 640.511,A -85,B 0,C 180,E1 -10916.87,E2 -10916.87} C_VEL
LIN {X 0,Y 417.408,Z 624.183,A -85,B 0,C 180,E1 -10917.751,E2 -10917.751} C_VEL
LIN {X 0,Y 417.954,Z 617.017,A -85,B 0,C 180,E1 -10918.089,E2 -10918.089} C_VEL
LIN {X 0,Y 414.338,Z 598.375,A -85,B 0,C 180,E1 -10919.315,E2 -10919.315} C_VEL
LIN {X 0,Y 411.381,Z 580.816,A -85,B 0,C 180,E1 -10920.314,E2 -10920.314} C_VEL
LIN {X 0,Y 408.586,Z 569.436,A -85,B 0,C 180,E1 -10920.997,E2 -10920.997} C_VEL
LIN {X 0,Y 406.596,Z 561.525,A -85,B 0,C 180,E1 -10921.52,E2 -10921.52} C_VEL
LIN {X 0,Y 407.215,Z 550.355,A -85,B 0,C 180,E1 -10924.719,E2 -10924.719} C_VEL
LIN {X 0,Y 407.853,Z 540.963,A -85,B 0,C 180,E1 -10927.566,E2 -10927.566} C_VEL
LIN {X 0,Y 408.544,Z 532.983,A -85,B 0,C 180,E1 -10930.174,E2 -10930.174} C_VEL
LIN {X 0,Y 408.396,Z 529.399,A -85,B 0,C 180,E1 -10931.494,E2 -10931.494} C_VEL
LIN {X 0,Y 407.589,Z 524.377,A -85,B 0,C 180,E1 -10933.608,E2 -10933.608} C_VEL
LIN {X 0,Y 406.598,Z 519.182,A -85,B 0,C 180,E1 -10936.26,E2 -10936.26} C_VEL
LIN {X 0,Y 405.714,Z 515.396,A -85,B 0,C 180,E1 -10938.833,E2 -10938.833} C_VEL
LIN {X 0,Y 405.15,Z 512.772,A -85,B 0,C 180,E1 -10941.356,E2 -10941.356} C_VEL
LIN {X 0,Y 404.738,Z 511.184,A -85,B 0,C 180,E1 -10943.816,E2 -10943.816} C_VEL
LIN {X 0,Y 404.532,Z 510.316,A -85,B 0,C 180,E1 -10946.503,E2 -10946.503} C_VEL
LIN {X 0,Y 404.498,Z 510.176,A -85,B 0,C 180,E1 -10948.948,E2 -10948.948} C_VEL
LIN {X 0,Y 406.019,Z 512.854,A -85,B 0,C 180,E1 -10949.272,E2 -10949.272} C_VEL
LIN {X 0,Y 407.3,Z 514.603,A -85,B 0,C 180,E1 -10949.509,E2 -10949.509} C_VEL
LIN {X 0,Y 410.988,Z 520.885,A -85,B 0,C 180,E1 -10950.234,E2 -10950.234} C_VEL
LIN {X 0,Y 416.071,Z 531.562,A -85,B 0,C 180,E1 -10951.318,E2 -10951.318} C_VEL
LIN {X 0,Y 419.469,Z 541.114,A -85,B 0,C 180,E1 -10952.189,E2 -10952.189} C_VEL
LIN {X 0,Y 417.951,Z 557.894,A -85,B 0,C 180,E1 -10953.153,E2 -10953.153} C_VEL
LIN {X 0,Y 416.334,Z 573.214,A -85,B 0,C 180,E1 -10954.236,E2 -10954.236} C_VEL
LIN {X 0,Y 414.733,Z 587.553,A -85,B 0,C 180,E1 -10955.47,E2 -10955.47} C_VEL
LIN {X 0,Y 412.967,Z 602.024,A -85,B 0,C 180,E1 -10956.957,E2 -10956.957} C_VEL
LIN {X 0,Y 411.348,Z 614.239,A -85,B 0,C 180,E1 -10958.449,E2 -10958.449} C_VEL
LIN {X 0,Y 409.764,Z 626.348,A -85,B 0,C 180,E1 -10960.201,E2 -10960.201} C_VEL
LIN {X 0,Y 408.288,Z 636.625,A -85,B 0,C 180,E1 -10961.951,E2 -10961.951} C_VEL
LIN {X 0,Y 406.913,Z 646.466,A -85,B 0,C 180,E1 -10963.958,E2 -10963.958} C_VEL
LIN {X 0,Y 405.866,Z 654.625,A -85,B 0,C 180,E1 -10965.971,E2 -10965.971} C_VEL
LIN {X 0,Y 404.991,Z 661.355,A -85,B 0,C 180,E1 -10967.981,E2 -10967.981} C_VEL
LIN {X 0,Y 404.45,Z 666.856,A -85,B 0,C 180,E1 -10969.994,E2 -10969.994} C_VEL
LIN {X 0,Y 403.981,Z 671.15,A -85,B 0,C 180,E1 -10972,E2 -10972} C_VEL
LIN {X 0,Y 403.727,Z 674.367,A -85,B 0,C 180,E1 -10974.005,E2 -10974.005} C_VEL
LIN {X 0,Y 403.496,Z 676.603,A -85,B 0,C 180,E1 -10976.005,E2 -10976.005} C_VEL
LIN {X 0,Y 403.263,Z 677.823,A -85,B 0,C 180,E1 -10978.003,E2 -10978.003} C_VEL
LIN {X 0,Y 403.161,Z 678.148,A -85,B 0,C 180,E1 -10980,E2 -10980} C_VEL
LIN {X 0,Y 403.227,Z 677.417,A -85,B 0,C 180,E1 -10981.998,E2 -10981.998} C_VEL
LIN {X 0,Y 403.478,Z 675.787,A -85,B 0,C 180,E1 -10983.996,E2 -10983.996} C_VEL
LIN {X 0,Y 403.418,Z 673.138,A -85,B 0,C 180,E1 -10986,E2 -10986} C_VEL
LIN {X 0,Y 403.74,Z 669.475,A -85,B 0,C 180,E1 -10988.005,E2 -10988.005} C_VEL
LIN {X 0,Y 404.045,Z 664.717,A -85,B 0,C 180,E1 -10990.018,E2 -10990.018} C_VEL
LIN {X 0,Y 404.517,Z 658.761,A -85,B 0,C 180,E1 -10992.034,E2 -10992.034} C_VEL
LIN {X 0,Y 405.309,Z 651.522,A -85,B 0,C 180,E1 -10994.05,E2 -10994.05} C_VEL
LIN {X 0,Y 406.283,Z 642.82,A -85,B 0,C 180,E1 -10996.068,E2 -10996.068} C_VEL
LIN {X 0,Y 407.53,Z 632.363,A -85,B 0,C 180,E1 -10998.085,E2 -10998.085} C_VEL
LIN {X 0,Y 408.79,Z 621.522,A -85,B 0,C 180,E1 -10999.85,E2 -10999.85} C_VEL
LIN {X 0,Y 410.388,Z 608.769,A -85,B 0,C 180,E1 -11001.605,E2 -11001.605} C_VEL
LIN {X 0,Y 411.915,Z 595.891,A -85,B 0,C 180,E1 -11003.106,E2 -11003.106} C_VEL
LIN {X 0,Y 413.483,Z 582.002,A -85,B 0,C 180,E1 -11004.476,E2 -11004.476} C_VEL
LIN {X 0,Y 414.991,Z 568.577,A -85,B 0,C 180,E1 -11005.586,E2 -11005.586} C_VEL
LIN {X 0,Y 416.129,Z 555.15,A -85,B 0,C 180,E1 -11006.529,E2 -11006.529} C_VEL
LIN {X 0,Y 417.391,Z 540.4,A -85,B 0,C 180,E1 -11007.382,E2 -11007.382} C_VEL
LIN {X 0,Y 413.387,Z 529.698,A -85,B 0,C 180,E1 -11008.214,E2 -11008.214} C_VEL
LIN {X 0,Y 406.078,Z 513.289,A -85,B 0,C 180,E1 -11009.42,E2 -11009.42} C_VEL
LIN {X 0,Y 404.271,Z 508.988,A -85,B 0,C 180,E1 -11009.705,E2 -11009.705} C_VEL
LIN {X 0,Y 404.175,Z 508.453,A -85,B 0,C 180,E1 -11009.754,E2 -11009.754} C_VEL
LIN {X 0,Y 404.176,Z 508.454,A -85,B 0,C 180,E1 -11013.42,E2 -11013.42} C_VEL
LIN {X 0,Y 404.149,Z 508.457,A -85,B 0,C 180,E1 -11016.246,E2 -11016.246} C_VEL
LIN {X 0,Y 404.161,Z 508.455,A -85,B 0,C 180,E1 -11018.757,E2 -11018.757} C_VEL
LIN {X 0,Y 404.128,Z 508.459,A -85,B 0,C 180,E1 -11021.6,E2 -11021.6} C_VEL
LIN {X 0,Y 404.15,Z 508.458,A -85,B 0,C 180,E1 -11024.522,E2 -11024.522} C_VEL
LIN {X 0,Y 404.142,Z 508.457,A -85,B 0,C 180,E1 -11027.296,E2 -11027.296} C_VEL
LIN {X 0,Y 404.175,Z 508.453,A -85,B 0,C 180,E1 -11029.955,E2 -11029.955} C_VEL
LIN {X 0,Y 404.142,Z 508.456,A -85,B 0,C 180,E1 -11033.125,E2 -11033.125} C_VEL
LIN {X 0,Y 404.151,Z 508.462,A -85,B 0,C 180,E1 -11036.187,E2 -11036.187} C_VEL
LIN {X 0,Y 404.152,Z 508.46,A -85,B 0,C 180,E1 -11039.715,E2 -11039.715} C_VEL
LIN {X 0,Y 404.256,Z 508.545,A -85,B 0,C 180,E1 -11042.812,E2 -11042.812} C_VEL
LIN {X 0,Y 404.78,Z 512.8,A -85,B 0,C 180,E1 -11045.373,E2 -11045.373} C_VEL
LIN {X 0,Y 404.781,Z 518.26,A -85,B 0,C 180,E1 -11048.615,E2 -11048.615} C_VEL
LIN {X 0,Y 404.67,Z 523.578,A -85,B 0,C 180,E1 -11051.783,E2 -11051.783} C_VEL
LIN {X 0,Y 404.593,Z 528.18,A -85,B 0,C 180,E1 -11054.582,E2 -11054.582} C_VEL
LIN {X 0,Y 406.635,Z 533.603,A -85,B 0,C 180,E1 -11054.851,E2 -11054.851} C_VEL
LIN {X 0,Y 413.256,Z 550.19,A -85,B 0,C 180,E1 -11055.783,E2 -11055.783} C_VEL
LIN {X 0,Y 418.796,Z 566.393,A -85,B 0,C 180,E1 -11056.81,E2 -11056.81} C_VEL
LIN {X 0,Y 419.034,Z 568.251,A -85,B 0,C 180,E1 -11056.913,E2 -11056.913} C_VEL
LIN {X 0,Y 417.914,Z 583.455,A -85,B 0,C 180,E1 -11057.649,E2 -11057.649} C_VEL
LIN {X 0,Y 416.542,Z 598.499,A -85,B 0,C 180,E1 -11058.565,E2 -11058.565} C_VEL
LIN {X 0,Y 414.87,Z 614.191,A -85,B 0,C 180,E1 -11059.753,E2 -11059.753} C_VEL
LIN {X 0,Y 413.163,Z 628.399,A -85,B 0,C 180,E1 -11061.07,E2 -11061.07} C_VEL
LIN {X 0,Y 411.525,Z 641.162,A -85,B 0,C 180,E1 -11062.484,E2 -11062.484} C_VEL
LIN {X 0,Y 409.823,Z 653.491,A -85,B 0,C 180,E1 -11064.093,E2 -11064.093} C_VEL
LIN {X 0,Y 408.299,Z 664.593,A -85,B 0,C 180,E1 -11065.804,E2 -11065.804} C_VEL
LIN {X 0,Y 407.232,Z 672.079,A -85,B 0,C 180,E1 -11067.142,E2 -11067.142} C_VEL
LIN {X 0,Y 406.078,Z 675.62,A -85,B 0,C 180,E1 -11067.793,E2 -11067.793} C_VEL
LIN {X 0,Y 399.669,Z 685.438,A -85,B 0,C 180,E1 -11069.711,E2 -11069.711} C_VEL
LIN {X 0,Y 398.281,Z 688.368,A -85,B 0,C 180,E1 -11070.418,E2 -11070.418} C_VEL
LIN {X 0,Y 398.078,Z 689.301,A -85,B 0,C 180,E1 -11070.665,E2 -11070.665} C_VEL
LIN {X 0,Y 397.29,Z 695.634,A -85,B 0,C 180,E1 -11072.534,E2 -11072.534} C_VEL
LIN {X 0,Y 396.776,Z 701.379,A -85,B 0,C 180,E1 -11074.571,E2 -11074.571} C_VEL
LIN {X 0,Y 396.265,Z 706.973,A -85,B 0,C 180,E1 -11077.13,E2 -11077.13} C_VEL
LIN {X 0,Y 395.965,Z 710.243,A -85,B 0,C 180,E1 -11079.191,E2 -11079.191} C_VEL
LIN {X 0,Y 395.85,Z 712.577,A -85,B 0,C 180,E1 -11081.261,E2 -11081.261} C_VEL
LIN {X 0,Y 395.739,Z 713.896,A -85,B 0,C 180,E1 -11083.347,E2 -11083.347} C_VEL
LIN {X 0,Y 395.7,Z 714.257,A -85,B 0,C 180,E1 -11085.45,E2 -11085.45} C_VEL
LIN {X 0,Y 395.707,Z 713.626,A -85,B 0,C 180,E1 -11087.572,E2 -11087.572} C_VEL
LIN {X 0,Y 395.826,Z 711.864,A -85,B 0,C 180,E1 -11089.773,E2 -11089.773} C_VEL
LIN {X 0,Y 396.081,Z 709.206,A -85,B 0,C 180,E1 -11091.876,E2 -11091.876} C_VEL
LIN {X 0,Y 396.486,Z 705.249,A -85,B 0,C 180,E1 -11094.058,E2 -11094.058} C_VEL
LIN {X 0,Y 397.066,Z 700.063,A -85,B 0,C 180,E1 -11096.262,E2 -11096.262} C_VEL
LIN {X 0,Y 397.837,Z 693.516,A -85,B 0,C 180,E1 -11098.486,E2 -11098.486} C_VEL
LIN {X 0,Y 398.96,Z 685.411,A -85,B 0,C 180,E1 -11100.719,E2 -11100.719} C_VEL
LIN {X 0,Y 400.2,Z 676.91,A -85,B 0,C 180,E1 -11102.655,E2 -11102.655} C_VEL
LIN {X 0,Y 401.604,Z 667.87,A -85,B 0,C 180,E1 -11104.405,E2 -11104.405} C_VEL
LIN {X 0,Y 403.206,Z 658.135,A -85,B 0,C 180,E1 -11106.033,E2 -11106.033} C_VEL
LIN {X 0,Y 405.113,Z 645.257,A -85,B 0,C 180,E1 -11107.855,E2 -11107.855} C_VEL
LIN {X 0,Y 407.145,Z 631.799,A -85,B 0,C 180,E1 -11109.433,E2 -11109.433} C_VEL
LIN {X 0,Y 408.984,Z 618.223,A -85,B 0,C 180,E1 -11110.766,E2 -11110.766} C_VEL
LIN {X 0,Y 410.845,Z 603.054,A -85,B 0,C 180,E1 -11111.998,E2 -11111.998} C_VEL
LIN {X 0,Y 412.424,Z 588.41,A -85,B 0,C 180,E1 -11112.969,E2 -11112.969} C_VEL
LIN {X 0,Y 413.788,Z 572.4,A -85,B 0,C 180,E1 -11113.817,E2 -11113.817} C_VEL
LIN {X 0,Y 413.815,Z 569.574,A -85,B 0,C 180,E1 -11113.953,E2 -11113.953} C_VEL
LIN {X 0,Y 409.421,Z 555.761,A -85,B 0,C 180,E1 -11114.964,E2 -11114.964} C_VEL
LIN {X 0,Y 403.083,Z 540.596,A -85,B 0,C 180,E1 -11116.039,E2 -11116.039} C_VEL
LIN {X 0,Y 398.171,Z 530.415,A -85,B 0,C 180,E1 -11116.758,E2 -11116.758} C_VEL
LIN {X 0,Y 397.976,Z 529.531,A -85,B 0,C 180,E1 -11116.819,E2 -11116.819} C_VEL
LIN {X 0,Y 398.115,Z 525.477,A -85,B 0,C 180,E1 -11119.381,E2 -11119.381} C_VEL
LIN {X 0,Y 398.267,Z 520.428,A -85,B 0,C 180,E1 -11122.567,E2 -11122.567} C_VEL
LIN {X 0,Y 398.32,Z 517.507,A -85,B 0,C 180,E1 -11124.39,E2 -11124.39} C_VEL
LIN {X 0,Y 397.939,Z 513.862,A -85,B 0,C 180,E1 -11126.804,E2 -11126.804} C_VEL
LIN {X 0,Y 397.129,Z 509.336,A -85,B 0,C 180,E1 -11129.752,E2 -11129.752} C_VEL
LIN {X 0,Y 397.187,Z 509.324,A -85,B 0,C 180,E1 -11132.609,E2 -11132.609} C_VEL
LIN {X 0,Y 397.125,Z 509.334,A -85,B 0,C 180,E1 -11135.981,E2 -11135.981} C_VEL
LIN {X 0,Y 397.145,Z 509.33,A -85,B 0,C 180,E1 -11139.697,E2 -11139.697} C_VEL
LIN {X 0,Y 397.172,Z 509.324,A -85,B 0,C 180,E1 -11142.844,E2 -11142.844} C_VEL
LIN {X 0,Y 397.216,Z 509.316,A -85,B 0,C 180,E1 -11146.678,E2 -11146.678} C_VEL
LIN {X 0,Y 397.219,Z 509.317,A -85,B 0,C 180,E1 -11149.809,E2 -11149.809} C_VEL
LIN {X 0,Y 397.355,Z 509.301,A -85,B 0,C 180,E1 -11152.888,E2 -11152.888} C_VEL
LIN {X 0,Y 397.253,Z 509.309,A -85,B 0,C 180,E1 -11154.925,E2 -11154.925} C_VEL
LIN {X 0,Y 397.442,Z 509.285,A -85,B 0,C 180,E1 -11157.973,E2 -11157.973} C_VEL
LIN {X 0,Y 397.572,Z 509.275,A -85,B 0,C 180,E1 -11160,E2 -11160} C_VEL
LIN {X 0,Y 397.373,Z 509.297,A -85,B 0,C 180,E1 -11163.041,E2 -11163.041} C_VEL
LIN {X 0,Y 397.353,Z 509.301,A -85,B 0,C 180,E1 -11167.112,E2 -11167.112} C_VEL
LIN {X 0,Y 397.219,Z 509.316,A -85,B 0,C 180,E1 -11170.191,E2 -11170.191} C_VEL
LIN {X 0,Y 397.215,Z 509.315,A -85,B 0,C 180,E1 -11173.321,E2 -11173.321} C_VEL
LIN {X 0,Y 397.17,Z 509.29,A -85,B 0,C 180,E1 -11177.155,E2 -11177.155} C_VEL
LIN {X 0,Y 397.145,Z 509.327,A -85,B 0,C 180,E1 -11180.727,E2 -11180.727} C_VEL
LIN {X 0,Y 397.129,Z 509.298,A -85,B 0,C 180,E1 -11184.018,E2 -11184.018} C_VEL
LIN {X 0,Y 397.184,Z 509.323,A -85,B 0,C 180,E1 -11187.39,E2 -11187.39} C_VEL
LIN {X 0,Y 397.076,Z 509.337,A -85,B 0,C 180,E1 -11190.882,E2 -11190.882} C_VEL
LIN {X 0,Y 397.116,Z 509.33,A -85,B 0,C 180,E1 -11194.494,E2 -11194.494} C_VEL
LIN {X 0,Y 397.117,Z 509.388,A -85,B 0,C 180,E1 -11197.623,E2 -11197.623} C_VEL
LIN {X 0,Y 398.869,Z 517.118,A -85,B 0,C 180,E1 -11200.745,E2 -11200.745} C_VEL
LIN {X 0,Y 400.707,Z 525.655,A -85,B 0,C 180,E1 -11204.022,E2 -11204.022} C_VEL
LIN {X 0,Y 402.554,Z 534.22,A -85,B 0,C 180,E1 -11207.16,E2 -11207.16} C_VEL
LIN {X 0,Y 403.185,Z 538.18,A -85,B 0,C 180,E1 -11208.55,E2 -11208.55} C_VEL
LIN {X 0,Y 402.831,Z 544.511,A -85,B 0,C 180,E1 -11210.601,E2 -11210.601} C_VEL
LIN {X 0,Y 401.979,Z 553.831,A -85,B 0,C 180,E1 -11213.536,E2 -11213.536} C_VEL
LIN {X 0,Y 401.086,Z 563.5,A -85,B 0,C 180,E1 -11216.5,E2 -11216.5} C_VEL
LIN {X 0,Y 400.459,Z 571.042,A -85,B 0,C 180,E1 -11218.731,E2 -11218.731} C_VEL
LIN {X 0,Y 406.628,Z 593.518,A -85,B 0,C 180,E1 -11219.857,E2 -11219.857} C_VEL
LIN {X 0,Y 410.455,Z 610.761,A -85,B 0,C 180,E1 -11220.837,E2 -11220.837} C_VEL
LIN {X 0,Y 412.069,Z 618.421,A -85,B 0,C 180,E1 -11221.327,E2 -11221.327} C_VEL
LIN {X 0,Y 410.673,Z 634.839,A -85,B 0,C 180,E1 -11222.205,E2 -11222.205} C_VEL
LIN {X 0,Y 408.919,Z 649.74,A -85,B 0,C 180,E1 -11223.184,E2 -11223.184} C_VEL
LIN {X 0,Y 407.016,Z 665.198,A -85,B 0,C 180,E1 -11224.427,E2 -11224.427} C_VEL
LIN {X 0,Y 405.091,Z 679.451,A -85,B 0,C 180,E1 -11225.805,E2 -11225.805} C_VEL
LIN {X 0,Y 403.442,Z 691.688,A -85,B 0,C 180,E1 -11227.196,E2 -11227.196} C_VEL
LIN {X 0,Y 401.617,Z 704.912,A -85,B 0,C 180,E1 -11228.979,E2 -11228.979} C_VEL
LIN {X 0,Y 400.076,Z 716.147,A -85,B 0,C 180,E1 -11230.771,E2 -11230.771} C_VEL
LIN {X 0,Y 398.723,Z 727.084,A -85,B 0,C 180,E1 -11232.829,E2 -11232.829} C_VEL
LIN {X 0,Y 397.759,Z 735.252,A -85,B 0,C 180,E1 -11234.632,E2 -11234.632} C_VEL
LIN {X 0,Y 396.992,Z 743.565,A -85,B 0,C 180,E1 -11236.821,E2 -11236.821} C_VEL
LIN {X 0,Y 396.447,Z 749.602,A -85,B 0,C 180,E1 -11238.756,E2 -11238.756} C_VEL
LIN {X 0,Y 396.117,Z 754.914,A -85,B 0,C 180,E1 -11240.813,E2 -11240.813} C_VEL
LIN {X 0,Y 395.98,Z 759.016,A -85,B 0,C 180,E1 -11242.864,E2 -11242.864} C_VEL
LIN {X 0,Y 395.881,Z 762.063,A -85,B 0,C 180,E1 -11244.909,E2 -11244.909} C_VEL
LIN {X 0,Y 395.882,Z 764.029,A -85,B 0,C 180,E1 -11246.948,E2 -11246.948} C_VEL
LIN {X 0,Y 395.915,Z 764.987,A -85,B 0,C 180,E1 -11248.984,E2 -11248.984} C_VEL
LIN {X 0,Y 395.916,Z 764.901,A -85,B 0,C 180,E1 -11251.018,E2 -11251.018} C_VEL
LIN {X 0,Y 395.897,Z 763.782,A -85,B 0,C 180,E1 -11253.054,E2 -11253.054} C_VEL
LIN {X 0,Y 395.899,Z 761.631,A -85,B 0,C 180,E1 -11255.093,E2 -11255.093} C_VEL
LIN {X 0,Y 396.021,Z 758.432,A -85,B 0,C 180,E1 -11257.137,E2 -11257.137} C_VEL
LIN {X 0,Y 396.127,Z 754.307,A -85,B 0,C 180,E1 -11259.189,E2 -11259.189} C_VEL
LIN {X 0,Y 396.459,Z 749.034,A -85,B 0,C 180,E1 -11261.245,E2 -11261.245} C_VEL
LIN {X 0,Y 397.039,Z 742.571,A -85,B 0,C 180,E1 -11263.305,E2 -11263.305} C_VEL
LIN {X 0,Y 397.771,Z 734.742,A -85,B 0,C 180,E1 -11265.369,E2 -11265.369} C_VEL
LIN {X 0,Y 398.73,Z 726.582,A -85,B 0,C 180,E1 -11267.173,E2 -11267.173} C_VEL
LIN {X 0,Y 400.081,Z 715.628,A -85,B 0,C 180,E1 -11269.231,E2 -11269.231} C_VEL
LIN {X 0,Y 401.576,Z 704.315,A -85,B 0,C 180,E1 -11271.026,E2 -11271.026} C_VEL
LIN {X 0,Y 403.287,Z 691.994,A -85,B 0,C 180,E1 -11272.68,E2 -11272.68} C_VEL
LIN {X 0,Y 405.089,Z 678.515,A -85,B 0,C 180,E1 -11274.198,E2 -11274.198} C_VEL
LIN {X 0,Y 406.757,Z 665.241,A -85,B 0,C 180,E1 -11275.455,E2 -11275.455} C_VEL
LIN {X 0,Y 408.426,Z 651.097,A -85,B 0,C 180,E1 -11276.578,E2 -11276.578} C_VEL
LIN {X 0,Y 410.03,Z 635.861,A -85,B 0,C 180,E1 -11277.568,E2 -11277.568} C_VEL
LIN {X 0,Y 411.535,Z 618.706,A -85,B 0,C 180,E1 -11278.45,E2 -11278.45} C_VEL
